LIN {X 0,Y 361.991,Z 217.011,A -85,B 0,C 180,E1 -12946.527,E2 -12946.527} C_VEL
LIN {X 0,Y 362.024,Z 217.007,A -85,B 0,C 180,E1 -12949.938,E2 -12949.938} C_VEL
LIN {X 0,Y 362.155,Z 216.995,A -85,B 0,C 180,E1 -12953.313,E2 -12953.313} C_VEL
LIN {X 0,Y 362.275,Z 216.981,A -85,B 0,C 180,E1 -12957.776,E2 -12957.776} C_VEL
LIN {X 0,Y 362.421,Z 216.956,A -85,B 0,C 180,E1 -12960,E2 -12960} C_VEL
LIN {X 0,Y 362.275,Z 216.984,A -85,B 0,C 180,E1 -12962.223,E2 -12962.223} C_VEL
LIN {X 0,Y 362.155,Z 217,A -85,B 0,C 180,E1 -12966.686,E2 -12966.686} C_VEL
LIN {X 0,Y 362.024,Z 217.013,A -85,B 0,C 180,E1 -12970.062,E2 -12970.062} C_VEL
LIN {X 0,Y 361.99,Z 217.014,A -85,B 0,C 180,E1 -12973.899,E2 -12973.899} C_VEL
LIN {X 0,Y 361.96,Z 217.016,A -85,B 0,C 180,E1 -12977.939,E2 -12977.939} C_VEL
LIN {X 0,Y 361.885,Z 217.026,A -85,B 0,C 180,E1 -12981.653,E2 -12981.653} C_VEL
LIN {X 0,Y 361.921,Z 217.022,A -85,B 0,C 180,E1 -12985.29,E2 -12985.29} C_VEL
LIN {X 0,Y 361.916,Z 217.03,A -85,B 0,C 180,E1 -12987.778,E2 -12987.778} C_VEL
LIN {X 0,Y 361.853,Z 217.036,A -85,B 0,C 180,E1 -12991.628,E2 -12991.628} C_VEL
LIN {X 0,Y 361.868,Z 217.032,A -85,B 0,C 180,E1 -12995.345,E2 -12995.345} C_VEL
LIN {X 0,Y 361.864,Z 217.028,A -85,B 0,C 180,E1 -12999.027,E2 -12999.027} C_VEL
LIN {X 0,Y 361.831,Z 217.039,A -85,B 0,C 180,E1 -13002.829,E2 -13002.829} C_VEL
LIN {X 0,Y 361.821,Z 217.04,A -85,B 0,C 180,E1 -13005.946,E2 -13005.946} C_VEL
LIN {X 0,Y 361.869,Z 217.033,A -85,B 0,C 180,E1 -13009.238,E2 -13009.238} C_VEL
LIN {X 0,Y 361.862,Z 217.11,A -85,B 0,C 180,E1 -13012.901,E2 -13012.901} C_VEL
LIN {X 0,Y 365.155,Z 229.037,A -85,B 0,C 180,E1 -13015.853,E2 -13015.853} C_VEL
LIN {X 0,Y 367.968,Z 240.182,A -85,B 0,C 180,E1 -13018.43,E2 -13018.43} C_VEL
LIN {X 0,Y 374.958,Z 256.162,A -85,B 0,C 180,E1 -13019.427,E2 -13019.427} C_VEL
LIN {X 0,Y 380.018,Z 282.754,A -85,B 0,C 180,E1 -13020.44,E2 -13020.44} C_VEL
LIN {X 0,Y 377.652,Z 382.363,A -85,B 0,C 180,E1 -13022.35,E2 -13022.35} C_VEL
LIN {X 0,Y 376.822,Z 408.501,A -85,B 0,C 180,E1 -13022.886,E2 -13022.886} C_VEL
LIN {X 0,Y 375.878,Z 423.941,A -85,B 0,C 180,E1 -13023.413,E2 -13023.413} C_VEL
LIN {X 0,Y 374.672,Z 437.728,A -85,B 0,C 180,E1 -13024.07,E2 -13024.07} C_VEL
LIN {X 0,Y 373.299,Z 451.151,A -85,B 0,C 180,E1 -13024.913,E2 -13024.913} C_VEL
LIN {X 0,Y 371.548,Z 464.972,A -85,B 0,C 180,E1 -13026.004,E2 -13026.004} C_VEL
LIN {X 0,Y 369.648,Z 478.71,A -85,B 0,C 180,E1 -13027.356,E2 -13027.356} C_VEL
LIN {X 0,Y 367.728,Z 491.149,A -85,B 0,C 180,E1 -13028.855,E2 -13028.855} C_VEL
LIN {X 0,Y 366.079,Z 502.385,A -85,B 0,C 180,E1 -13030.499,E2 -13030.499} C_VEL
LIN {X 0,Y 364.428,Z 512.768,A -85,B 0,C 180,E1 -13032.318,E2 -13032.318} C_VEL
LIN {X 0,Y 363.095,Z 522.038,A -85,B 0,C 180,E1 -13034.278,E2 -13034.278} C_VEL
LIN {X 0,Y 361.936,Z 530.768,A -85,B 0,C 180,E1 -13036.526,E2 -13036.526} C_VEL
LIN {X 0,Y 361.133,Z 537.778,A -85,B 0,C 180,E1 -13038.778,E2 -13038.778} C_VEL
LIN {X 0,Y 360.628,Z 543.293,A -85,B 0,C 180,E1 -13041.031,E2 -13041.031} C_VEL
LIN {X 0,Y 360.386,Z 547.465,A -85,B 0,C 180,E1 -13043.281,E2 -13043.281} C_VEL
LIN {X 0,Y 360.299,Z 550.391,A -85,B 0,C 180,E1 -13045.525,E2 -13045.525} C_VEL
LIN {X 0,Y 360.254,Z 552.136,A -85,B 0,C 180,E1 -13047.764,E2 -13047.764} C_VEL
LIN {X 0,Y 360.357,Z 552.736,A -85,B 0,C 180,E1 -13050,E2 -13050} C_VEL
LIN {X 0,Y 360.255,Z 552.129,A -85,B 0,C 180,E1 -13052.236,E2 -13052.236} C_VEL
LIN {X 0,Y 360.3,Z 550.375,A -85,B 0,C 180,E1 -13054.475,E2 -13054.475} C_VEL
LIN {X 0,Y 360.386,Z 547.445,A -85,B 0,C 180,E1 -13056.719,E2 -13056.719} C_VEL
LIN {X 0,Y 360.628,Z 543.272,A -85,B 0,C 180,E1 -13058.969,E2 -13058.969} C_VEL
LIN {X 0,Y 361.132,Z 537.746,A -85,B 0,C 180,E1 -13061.222,E2 -13061.222} C_VEL
LIN {X 0,Y 361.906,Z 530.719,A -85,B 0,C 180,E1 -13063.475,E2 -13063.475} C_VEL
LIN {X 0,Y 363.096,Z 521.982,A -85,B 0,C 180,E1 -13065.722,E2 -13065.722} C_VEL
LIN {X 0,Y 364.436,Z 512.704,A -85,B 0,C 180,E1 -13067.682,E2 -13067.682} C_VEL
LIN {X 0,Y 365.907,Z 503.649,A -85,B 0,C 180,E1 -13069.284,E2 -13069.284} C_VEL
LIN {X 0,Y 367.612,Z 492.084,A -85,B 0,C 180,E1 -13071.005,E2 -13071.005} C_VEL
LIN {X 0,Y 369.463,Z 479.824,A -85,B 0,C 180,E1 -13072.508,E2 -13072.508} C_VEL
LIN {X 0,Y 371.154,Z 467.779,A -85,B 0,C 180,E1 -13073.726,E2 -13073.726} C_VEL
LIN {X 0,Y 372.912,Z 454.014,A -85,B 0,C 180,E1 -13074.865,E2 -13074.865} C_VEL
LIN {X 0,Y 374.41,Z 440.215,A -85,B 0,C 180,E1 -13075.771,E2 -13075.771} C_VEL
LIN {X 0,Y 375.675,Z 425.49,A -85,B 0,C 180,E1 -13076.513,E2 -13076.513} C_VEL
LIN {X 0,Y 376.707,Z 410.344,A -85,B 0,C 180,E1 -13077.048,E2 -13077.048} C_VEL
LIN {X 0,Y 377.405,Z 390.605,A -85,B 0,C 180,E1 -13077.482,E2 -13077.482} C_VEL
LIN {X 0,Y 380.074,Z 283.543,A -85,B 0,C 180,E1 -13079.523,E2 -13079.523} C_VEL
LIN {X 0,Y 375.075,Z 256.666,A -85,B 0,C 180,E1 -13080.534,E2 -13080.534} C_VEL
LIN {X 0,Y 372.927,Z 251.228,A -85,B 0,C 180,E1 -13080.847,E2 -13080.847} C_VEL
LIN {X 0,Y 367.805,Z 239.811,A -85,B 0,C 180,E1 -13081.61,E2 -13081.61} C_VEL
LIN {X 0,Y 364.596,Z 226.834,A -85,B 0,C 180,E1 -13084.654,E2 -13084.654} C_VEL
LIN {X 0,Y 361.875,Z 217.034,A -85,B 0,C 180,E1 -13087.125,E2 -13087.125} C_VEL
LIN {X 0,Y 361.869,Z 217.034,A -85,B 0,C 180,E1 -13090.762,E2 -13090.762} C_VEL
LIN {X 0,Y 361.817,Z 217.039,A -85,B 0,C 180,E1 -13094.367,E2 -13094.367} C_VEL
LIN {X 0,Y 361.851,Z 217.031,A -85,B 0,C 180,E1 -13097.564,E2 -13097.564} C_VEL
LIN {X 0,Y 361.869,Z 217.029,A -85,B 0,C 180,E1 -13100.972,E2 -13100.972} C_VEL
LIN {X 0,Y 361.869,Z 217.026,A -85,B 0,C 180,E1 -13104.655,E2 -13104.655} C_VEL
LIN {X 0,Y 361.853,Z 217.033,A -85,B 0,C 180,E1 -13108.372,E2 -13108.372} C_VEL
LIN {X 0,Y 361.916,Z 217.025,A -85,B 0,C 180,E1 -13112.222,E2 -13112.222} C_VEL
LIN {X 0,Y 361.92,Z 217.026,A -85,B 0,C 180,E1 -13114.709,E2 -13114.709} C_VEL
LIN {X 0,Y 361.854,Z 217.011,A -85,B 0,C 180,E1 -13118.345,E2 -13118.345} C_VEL
LIN {X 0,Y 361.96,Z 217.022,A -85,B 0,C 180,E1 -13122.061,E2 -13122.061} C_VEL
LIN {X 0,Y 361.99,Z 217.017,A -85,B 0,C 180,E1 -13126.101,E2 -13126.101} C_VEL
LIN {X 0,Y 362.024,Z 217.014,A -85,B 0,C 180,E1 -13129.938,E2 -13129.938} C_VEL
LIN {X 0,Y 362.155,Z 216.999,A -85,B 0,C 180,E1 -13133.314,E2 -13133.314} C_VEL
LIN {X 0,Y 362.275,Z 216.984,A -85,B 0,C 180,E1 -13137.777,E2 -13137.777} C_VEL
LIN {X 0,Y 362.421,Z 216.957,A -85,B 0,C 180,E1 -13140,E2 -13140} C_VEL
LIN {X 0,Y 362.275,Z 216.982,A -85,B 0,C 180,E1 -13142.224,E2 -13142.224} C_VEL
LIN {X 0,Y 362.157,Z 216.997,A -85,B 0,C 180,E1 -13146.687,E2 -13146.687} C_VEL
LIN {X 0,Y 362.024,Z 217.013,A -85,B 0,C 180,E1 -13150.062,E2 -13150.062} C_VEL
LIN {X 0,Y 361.991,Z 217.017,A -85,B 0,C 180,E1 -13153.899,E2 -13153.899} C_VEL
LIN {X 0,Y 361.961,Z 217.02,A -85,B 0,C 180,E1 -13157.939,E2 -13157.939} C_VEL
LIN {X 0,Y 361.855,Z 217.035,A -85,B 0,C 180,E1 -13161.655,E2 -13161.655} C_VEL
LIN {X 0,Y 361.921,Z 217.004,A -85,B 0,C 180,E1 -13165.291,E2 -13165.291} C_VEL
LIN {X 0,Y 361.917,Z 217.022,A -85,B 0,C 180,E1 -13167.778,E2 -13167.778} C_VEL
LIN {X 0,Y 361.841,Z 217.035,A -85,B 0,C 180,E1 -13171.286,E2 -13171.286} C_VEL
LIN {X 0,Y 361.849,Z 217.03,A -85,B 0,C 180,E1 -13174.281,E2 -13174.281} C_VEL
LIN {X 0,Y 361.86,Z 217.032,A -85,B 0,C 180,E1 -13177.224,E2 -13177.224} C_VEL
LIN {X 0,Y 361.832,Z 217.038,A -85,B 0,C 180,E1 -13180.756,E2 -13180.756} C_VEL
LIN {X 0,Y 361.832,Z 217.035,A -85,B 0,C 180,E1 -13184.366,E2 -13184.366} C_VEL
LIN {X 0,Y 361.834,Z 217.038,A -85,B 0,C 180,E1 -13187.569,E2 -13187.569} C_VEL
LIN {X 0,Y 361.867,Z 217.027,A -85,B 0,C 180,E1 -13190.974,E2 -13190.974} C_VEL
LIN {X 0,Y 361.872,Z 217.029,A -85,B 0,C 180,E1 -13194.656,E2 -13194.656} C_VEL
LIN {X 0,Y 361.886,Z 217.145,A -85,B 0,C 180,E1 -13196.515,E2 -13196.515} C_VEL
LIN {X 0,Y 363.49,Z 223.101,A -85,B 0,C 180,E1 -13198.071,E2 -13198.071} C_VEL
LIN {X 0,Y 373.982,Z 244.423,A -85,B 0,C 180,E1 -13199.543,E2 -13199.543} C_VEL
LIN {X 0,Y 380.458,Z 259.445,A -85,B 0,C 180,E1 -13200.441,E2 -13200.441} C_VEL
LIN {X 0,Y 378.098,Z 358.781,A -85,B 0,C 180,E1 -13202.348,E2 -13202.348} C_VEL
LIN {X 0,Y 377.231,Z 388.834,A -85,B 0,C 180,E1 -13202.955,E2 -13202.955} C_VEL
LIN {X 0,Y 376.427,Z 403.824,A -85,B 0,C 180,E1 -13203.46,E2 -13203.46} C_VEL
LIN {X 0,Y 375.345,Z 418.287,A -85,B 0,C 180,E1 -13204.156,E2 -13204.156} C_VEL
LIN {X 0,Y 373.919,Z 433.412,A -85,B 0,C 180,E1 -13205.131,E2 -13205.131} C_VEL
LIN {X 0,Y 372.357,Z 446.659,A -85,B 0,C 180,E1 -13206.207,E2 -13206.207} C_VEL
LIN {X 0,Y 370.485,Z 460.122,A -85,B 0,C 180,E1 -13207.557,E2 -13207.557} C_VEL
LIN {X 0,Y 368.608,Z 472.69,A -85,B 0,C 180,E1 -13209.108,E2 -13209.108} C_VEL
LIN {X 0,Y 366.973,Z 483.449,A -85,B 0,C 180,E1 -13210.71,E2 -13210.71} C_VEL
LIN {X 0,Y 365.256,Z 494.245,A -85,B 0,C 180,E1 -13212.648,E2 -13212.648} C_VEL
LIN {X 0,Y 363.79,Z 503.32,A -85,B 0,C 180,E1 -13214.624,E2 -13214.624} C_VEL
LIN {X 0,Y 362.785,Z 510.621,A -85,B 0,C 180,E1 -13216.558,E2 -13216.558} C_VEL
LIN {X 0,Y 361.722,Z 517.558,A -85,B 0,C 180,E1 -13218.797,E2 -13218.797} C_VEL
LIN {X 0,Y 361.116,Z 523.003,A -85,B 0,C 180,E1 -13221.043,E2 -13221.043} C_VEL
LIN {X 0,Y 360.717,Z 527.515,A -85,B 0,C 180,E1 -13223.544,E2 -13223.544} C_VEL
LIN {X 0,Y 360.486,Z 530,A -85,B 0,C 180,E1 -13225.527,E2 -13225.527} C_VEL
LIN {X 0,Y 360.345,Z 531.738,A -85,B 0,C 180,E1 -13227.765,E2 -13227.765} C_VEL
LIN {X 0,Y 360.36,Z 532.344,A -85,B 0,C 180,E1 -13230,E2 -13230} C_VEL
LIN {X 0,Y 360.345,Z 531.784,A -85,B 0,C 180,E1 -13232.235,E2 -13232.235} C_VEL
LIN {X 0,Y 360.482,Z 530.106,A -85,B 0,C 180,E1 -13234.473,E2 -13234.473} C_VEL
LIN {X 0,Y 360.7,Z 527.276,A -85,B 0,C 180,E1 -13236.713,E2 -13236.713} C_VEL
LIN {X 0,Y 361.094,Z 523.222,A -85,B 0,C 180,E1 -13238.957,E2 -13238.957} C_VEL
LIN {X 0,Y 361.701,Z 517.846,A -85,B 0,C 180,E1 -13241.204,E2 -13241.204} C_VEL
LIN {X 0,Y 362.773,Z 510.986,A -85,B 0,C 180,E1 -13243.443,E2 -13243.443} C_VEL
LIN {X 0,Y 363.787,Z 503.616,A -85,B 0,C 180,E1 -13245.404,E2 -13245.404} C_VEL
LIN {X 0,Y 364.592,Z 498.483,A -85,B 0,C 180,E1 -13246.576,E2 -13246.576} C_VEL
LIN {X 0,Y 364.523,Z 495.062,A -85,B 0,C 180,E1 -13247.322,E2 -13247.322} C_VEL
LIN {X 0,Y 362.726,Z 489.389,A -85,B 0,C 180,E1 -13248.566,E2 -13248.566} C_VEL
LIN {X 0,Y 361.004,Z 483.3,A -85,B 0,C 180,E1 -13249.783,E2 -13249.783} C_VEL
LIN {X 0,Y 361.033,Z 479.222,A -85,B 0,C 180,E1 -13250.468,E2 -13250.468} C_VEL
LIN {X 0,Y 362.793,Z 467.979,A -85,B 0,C 180,E1 -13252.044,E2 -13252.044} C_VEL
LIN {X 0,Y 364.555,Z 456.112,A -85,B 0,C 180,E1 -13253.429,E2 -13253.429} C_VEL
LIN {X 0,Y 366.309,Z 443.263,A -85,B 0,C 180,E1 -13254.663,E2 -13254.663} C_VEL
LIN {X 0,Y 367.946,Z 429.165,A -85,B 0,C 180,E1 -13255.755,E2 -13255.755} C_VEL
LIN {X 0,Y 369.365,Z 413.988,A -85,B 0,C 180,E1 -13256.666,E2 -13256.666} C_VEL
LIN {X 0,Y 370.387,Z 399.264,A -85,B 0,C 180,E1 -13257.319,E2 -13257.319} C_VEL
LIN {X 0,Y 371.137,Z 384.589,A -85,B 0,C 180,E1 -13257.756,E2 -13257.756} C_VEL
LIN {X 0,Y 373.829,Z 283.961,A -85,B 0,C 180,E1 -13259.716,E2 -13259.716} C_VEL
LIN {X 0,Y 374.255,Z 261.257,A -85,B 0,C 180,E1 -13260.172,E2 -13260.172} C_VEL
LIN {X 0,Y 367.754,Z 246.374,A -85,B 0,C 180,E1 -13261.099,E2 -13261.099} C_VEL
LIN {X 0,Y 359.371,Z 229.462,A -85,B 0,C 180,E1 -13262.306,E2 -13262.306} C_VEL
LIN {X 0,Y 356.205,Z 223.066,A -85,B 0,C 180,E1 -13262.799,E2 -13262.799} C_VEL
LIN {X 0,Y 354.823,Z 217.911,A -85,B 0,C 180,E1 -13264.28,E2 -13264.28} C_VEL
LIN {X 0,Y 354.804,Z 217.92,A -85,B 0,C 180,E1 -13267.882,E2 -13267.882} C_VEL
LIN {X 0,Y 354.785,Z 217.918,A -85,B 0,C 180,E1 -13271.171,E2 -13271.171} C_VEL
LIN {X 0,Y 354.786,Z 217.914,A -85,B 0,C 180,E1 -13274.51,E2 -13274.51} C_VEL
LIN {X 0,Y 354.796,Z 217.901,A -85,B 0,C 180,E1 -13277.663,E2 -13277.663} C_VEL
LIN {X 0,Y 354.833,Z 217.91,A -85,B 0,C 180,E1 -13280.668,E2 -13280.668} C_VEL
LIN {X 0,Y 354.817,Z 217.907,A -85,B 0,C 180,E1 -13284.3,E2 -13284.3} C_VEL
LIN {X 0,Y 354.781,Z 217.898,A -85,B 0,C 180,E1 -13287.666,E2 -13287.666} C_VEL
LIN {X 0,Y 354.863,Z 217.9,A -85,B 0,C 180,E1 -13290.621,E2 -13290.621} C_VEL
LIN {X 0,Y 354.893,Z 217.897,A -85,B 0,C 180,E1 -13294.172,E2 -13294.172} C_VEL
LIN {X 0,Y 354.828,Z 217.905,A -85,B 0,C 180,E1 -13297.893,E2 -13297.893} C_VEL
LIN {X 0,Y 354.916,Z 217.893,A -85,B 0,C 180,E1 -13301.891,E2 -13301.891} C_VEL
LIN {X 0,Y 354.935,Z 217.887,A -85,B 0,C 180,E1 -13305.981,E2 -13305.981} C_VEL
LIN {X 0,Y 354.971,Z 217.885,A -85,B 0,C 180,E1 -13309.736,E2 -13309.736} C_VEL
LIN {X 0,Y 355.119,Z 217.872,A -85,B 0,C 180,E1 -13313.18,E2 -13313.18} C_VEL
LIN {X 0,Y 355.238,Z 217.858,A -85,B 0,C 180,E1 -13317.732,E2 -13317.732} C_VEL
LIN {X 0,Y 355.391,Z 217.832,A -85,B 0,C 180,E1 -13320,E2 -13320} C_VEL
LIN {X 0,Y 355.238,Z 217.861,A -85,B 0,C 180,E1 -13322.268,E2 -13322.268} C_VEL
LIN {X 0,Y 355.118,Z 217.875,A -85,B 0,C 180,E1 -13326.819,E2 -13326.819} C_VEL
LIN {X 0,Y 354.97,Z 217.893,A -85,B 0,C 180,E1 -13330.264,E2 -13330.264} C_VEL
LIN {X 0,Y 354.935,Z 217.894,A -85,B 0,C 180,E1 -13334.019,E2 -13334.019} C_VEL
LIN {X 0,Y 354.916,Z 217.895,A -85,B 0,C 180,E1 -13338.109,E2 -13338.109} C_VEL
LIN {X 0,Y 354.827,Z 217.906,A -85,B 0,C 180,E1 -13342.106,E2 -13342.106} C_VEL
LIN {X 0,Y 354.892,Z 217.897,A -85,B 0,C 180,E1 -13345.828,E2 -13345.828} C_VEL
LIN {X 0,Y 354.848,Z 217.909,A -85,B 0,C 180,E1 -13349.679,E2 -13349.679} C_VEL
LIN {X 0,Y 354.825,Z 217.906,A -85,B 0,C 180,E1 -13353.683,E2 -13353.683} C_VEL
LIN {X 0,Y 354.792,Z 217.911,A -85,B 0,C 180,E1 -13356.46,E2 -13356.46} C_VEL
LIN {X 0,Y 354.819,Z 217.899,A -85,B 0,C 180,E1 -13359.424,E2 -13359.424} C_VEL
LIN {X 0,Y 354.783,Z 217.917,A -85,B 0,C 180,E1 -13362.868,E2 -13362.868} C_VEL
LIN {X 0,Y 354.77,Z 217.917,A -85,B 0,C 180,E1 -13366.105,E2 -13366.105} C_VEL
LIN {X 0,Y 354.821,Z 217.911,A -85,B 0,C 180,E1 -13369.185,E2 -13369.185} C_VEL
LIN {X 0,Y 354.84,Z 218.074,A -85,B 0,C 180,E1 -13372.312,E2 -13372.312} C_VEL
LIN {X 0,Y 358.139,Z 229.843,A -85,B 0,C 180,E1 -13375.314,E2 -13375.314} C_VEL
LIN {X 0,Y 360.635,Z 239.833,A -85,B 0,C 180,E1 -13377.708,E2 -13377.708} C_VEL
LIN {X 0,Y 369.134,Z 258.831,A -85,B 0,C 180,E1 -13378.955,E2 -13378.955} C_VEL
LIN {X 0,Y 373.847,Z 283.787,A -85,B 0,C 180,E1 -13379.929,E2 -13379.929} C_VEL
LIN {X 0,Y 371.324,Z 383.972,A -85,B 0,C 180,E1 -13381.876,E2 -13381.876} C_VEL
LIN {X 0,Y 370.526,Z 408.314,A -85,B 0,C 180,E1 -13382.386,E2 -13382.386} C_VEL
LIN {X 0,Y 369.537,Z 423.747,A -85,B 0,C 180,E1 -13382.919,E2 -13382.919} C_VEL
LIN {X 0,Y 368.281,Z 437.523,A -85,B 0,C 180,E1 -13383.585,E2 -13383.585} C_VEL
LIN {X 0,Y 366.796,Z 451.504,A -85,B 0,C 180,E1 -13384.48,E2 -13384.48} C_VEL
LIN {X 0,Y 365.028,Z 464.774,A -85,B 0,C 180,E1 -13385.548,E2 -13385.548} C_VEL
LIN {X 0,Y 363.234,Z 477.216,A -85,B 0,C 180,E1 -13386.783,E2 -13386.783} C_VEL
LIN {X 0,Y 361.28,Z 489.877,A -85,B 0,C 180,E1 -13388.309,E2 -13388.309} C_VEL
LIN {X 0,Y 359.49,Z 500.912,A -85,B 0,C 180,E1 -13389.916,E2 -13389.916} C_VEL
LIN {X 0,Y 357.886,Z 511.075,A -85,B 0,C 180,E1 -13391.688,E2 -13391.688} C_VEL
LIN {X 0,Y 356.374,Z 520.597,A -85,B 0,C 180,E1 -13393.679,E2 -13393.679} C_VEL
LIN {X 0,Y 355.071,Z 529.307,A -85,B 0,C 180,E1 -13395.898,E2 -13395.898} C_VEL
LIN {X 0,Y 354.319,Z 535.951,A -85,B 0,C 180,E1 -13397.979,E2 -13397.979} C_VEL
LIN {X 0,Y 353.646,Z 541.836,A -85,B 0,C 180,E1 -13400.275,E2 -13400.275} C_VEL
LIN {X 0,Y 353.434,Z 545.339,A -85,B 0,C 180,E1 -13401.999,E2 -13401.999} C_VEL
LIN {X 0,Y 353.24,Z 548.878,A -85,B 0,C 180,E1 -13404.291,E2 -13404.291} C_VEL
LIN {X 0,Y 353.191,Z 551.208,A -85,B 0,C 180,E1 -13406.578,E2 -13406.578} C_VEL
LIN {X 0,Y 353.213,Z 552.38,A -85,B 0,C 180,E1 -13408.86,E2 -13408.86} C_VEL
LIN {X 0,Y 353.213,Z 552.377,A -85,B 0,C 180,E1 -13411.14,E2 -13411.14} C_VEL
LIN {X 0,Y 353.192,Z 551.195,A -85,B 0,C 180,E1 -13413.422,E2 -13413.422} C_VEL
LIN {X 0,Y 353.276,Z 548.603,A -85,B 0,C 180,E1 -13415.908,E2 -13415.908} C_VEL
LIN {X 0,Y 353.483,Z 544.241,A -85,B 0,C 180,E1 -13418.576,E2 -13418.576} C_VEL
LIN {X 0,Y 353.921,Z 539.043,A -85,B 0,C 180,E1 -13420.874,E2 -13420.874} C_VEL
LIN {X 0,Y 354.694,Z 532.401,A -85,B 0,C 180,E1 -13423.171,E2 -13423.171} C_VEL
LIN {X 0,Y 355.815,Z 524.128,A -85,B 0,C 180,E1 -13425.465,E2 -13425.465} C_VEL
LIN {X 0,Y 357.16,Z 515.309,A -85,B 0,C 180,E1 -13427.462,E2 -13427.462} C_VEL
LIN {X 0,Y 358.679,Z 506.352,A -85,B 0,C 180,E1 -13429.159,E2 -13429.159} C_VEL
LIN {X 0,Y 360.309,Z 495.798,A -85,B 0,C 180,E1 -13430.853,E2 -13430.853} C_VEL
LIN {X 0,Y 362.167,Z 484.331,A -85,B 0,C 180,E1 -13432.385,E2 -13432.385} C_VEL
LIN {X 0,Y 363.993,Z 471.866,A -85,B 0,C 180,E1 -13433.769,E2 -13433.769} C_VEL
LIN {X 0,Y 365.901,Z 458.218,A -85,B 0,C 180,E1 -13434.996,E2 -13434.996} C_VEL
LIN {X 0,Y 367.635,Z 443.594,A -85,B 0,C 180,E1 -13436.04,E2 -13436.04} C_VEL
LIN {X 0,Y 368.968,Z 429.525,A -85,B 0,C 180,E1 -13436.82,E2 -13436.82} C_VEL
LIN {X 0,Y 370.181,Z 413.557,A -85,B 0,C 180,E1 -13437.45,E2 -13437.45} C_VEL
LIN {X 0,Y 370.938,Z 397.546,A -85,B 0,C 180,E1 -13437.849,E2 -13437.849} C_VEL
LIN {X 0,Y 373.655,Z 292.386,A -85,B 0,C 180,E1 -13439.885,E2 -13439.885} C_VEL
LIN {X 0,Y 373.768,Z 283.974,A -85,B 0,C 180,E1 -13440.057,E2 -13440.057} C_VEL
LIN {X 0,Y 369.092,Z 258.68,A -85,B 0,C 180,E1 -13441.034,E2 -13441.034} C_VEL
LIN {X 0,Y 362.263,Z 243.483,A -85,B 0,C 180,E1 -13442.027,E2 -13442.027} C_VEL
LIN {X 0,Y 360.553,Z 239.569,A -85,B 0,C 180,E1 -13442.324,E2 -13442.324} C_VEL
LIN {X 0,Y 357.378,Z 226.863,A -85,B 0,C 180,E1 -13445.399,E2 -13445.399} C_VEL
LIN {X 0,Y 354.807,Z 217.915,A -85,B 0,C 180,E1 -13447.739,E2 -13447.739} C_VEL
LIN {X 0,Y 354.812,Z 217.911,A -85,B 0,C 180,E1 -13451.176,E2 -13451.176} C_VEL
LIN {X 0,Y 354.763,Z 217.916,A -85,B 0,C 180,E1 -13454.506,E2 -13454.506} C_VEL
LIN {X 0,Y 354.808,Z 217.909,A -85,B 0,C 180,E1 -13457.665,E2 -13457.665} C_VEL
LIN {X 0,Y 354.832,Z 217.906,A -85,B 0,C 180,E1 -13460.668,E2 -13460.668} C_VEL
LIN {X 0,Y 354.817,Z 217.904,A -85,B 0,C 180,E1 -13464.3,E2 -13464.3} C_VEL
LIN {X 0,Y 354.793,Z 217.909,A -85,B 0,C 180,E1 -13467.667,E2 -13467.667} C_VEL
LIN {X 0,Y 354.863,Z 217.901,A -85,B 0,C 180,E1 -13470.621,E2 -13470.621} C_VEL
LIN {X 0,Y 354.892,Z 217.903,A -85,B 0,C 180,E1 -13474.172,E2 -13474.172} C_VEL
LIN {X 0,Y 354.81,Z 217.889,A -85,B 0,C 180,E1 -13477.892,E2 -13477.892} C_VEL
LIN {X 0,Y 354.915,Z 217.901,A -85,B 0,C 180,E1 -13481.891,E2 -13481.891} C_VEL
LIN {X 0,Y 354.935,Z 217.896,A -85,B 0,C 180,E1 -13485.981,E2 -13485.981} C_VEL
LIN {X 0,Y 354.97,Z 217.894,A -85,B 0,C 180,E1 -13489.736,E2 -13489.736} C_VEL
LIN {X 0,Y 355.118,Z 217.874,A -85,B 0,C 180,E1 -13493.181,E2 -13493.181} C_VEL
LIN {X 0,Y 355.238,Z 217.861,A -85,B 0,C 180,E1 -13497.732,E2 -13497.732} C_VEL
LIN {X 0,Y 355.391,Z 217.833,A -85,B 0,C 180,E1 -13500,E2 -13500} C_VEL
LIN {X 0,Y 355.238,Z 217.858,A -85,B 0,C 180,E1 -13502.268,E2 -13502.268} C_VEL
LIN {X 0,Y 355.12,Z 217.875,A -85,B 0,C 180,E1 -13506.82,E2 -13506.82} C_VEL
LIN {X 0,Y 354.971,Z 217.891,A -85,B 0,C 180,E1 -13510.264,E2 -13510.264} C_VEL
LIN {X 0,Y 354.936,Z 217.895,A -85,B 0,C 180,E1 -13514.019,E2 -13514.019} C_VEL
LIN {X 0,Y 354.916,Z 217.898,A -85,B 0,C 180,E1 -13518.109,E2 -13518.109} C_VEL
LIN {X 0,Y 354.81,Z 217.911,A -85,B 0,C 180,E1 -13522.108,E2 -13522.108} C_VEL
LIN {X 0,Y 354.893,Z 217.876,A -85,B 0,C 180,E1 -13525.828,E2 -13525.828} C_VEL
LIN {X 0,Y 354.849,Z 217.907,A -85,B 0,C 180,E1 -13529.679,E2 -13529.679} C_VEL
LIN {X 0,Y 354.801,Z 217.908,A -85,B 0,C 180,E1 -13533.703,E2 -13533.703} C_VEL
LIN {X 0,Y 354.794,Z 217.912,A -85,B 0,C 180,E1 -13536.46,E2 -13536.46} C_VEL
LIN {X 0,Y 354.82,Z 217.906,A -85,B 0,C 180,E1 -13539.424,E2 -13539.424} C_VEL
LIN {X 0,Y 354.785,Z 217.915,A -85,B 0,C 180,E1 -13542.868,E2 -13542.868} C_VEL
LIN {X 0,Y 354.773,Z 217.916,A -85,B 0,C 180,E1 -13546.106,E2 -13546.106} C_VEL
LIN {X 0,Y 354.786,Z 217.919,A -85,B 0,C 180,E1 -13549.18,E2 -13549.18} C_VEL
LIN {X 0,Y 354.809,Z 217.915,A -85,B 0,C 180,E1 -13552.402,E2 -13552.402} C_VEL
LIN {X 0,Y 354.857,Z 218.081,A -85,B 0,C 180,E1 -13555.938,E2 -13555.938} C_VEL
LIN {X 0,Y 356.253,Z 223.233,A -85,B 0,C 180,E1 -13557.339,E2 -13557.339} C_VEL
LIN {X 0,Y 367.238,Z 245.255,A -85,B 0,C 180,E1 -13558.936,E2 -13558.936} C_VEL
LIN {X 0,Y 373.323,Z 258.985,A -85,B 0,C 180,E1 -13559.802,E2 -13559.802} C_VEL
LIN {X 0,Y 374.284,Z 261.371,A -85,B 0,C 180,E1 -13559.94,E2 -13559.94} C_VEL
LIN {X 0,Y 371.58,Z 369.725,A -85,B 0,C 180,E1 -13562.05,E2 -13562.05} C_VEL
LIN {X 0,Y 370.898,Z 390.19,A -85,B 0,C 180,E1 -13562.493,E2 -13562.493} C_VEL
LIN {X 0,Y 370.056,Z 404.688,A -85,B 0,C 180,E1 -13562.999,E2 -13562.999} C_VEL
LIN {X 0,Y 368.925,Z 419.126,A -85,B 0,C 180,E1 -13563.714,E2 -13563.714} C_VEL
LIN {X 0,Y 367.503,Z 433.618,A -85,B 0,C 180,E1 -13564.667,E2 -13564.667} C_VEL
LIN {X 0,Y 365.844,Z 446.866,A -85,B 0,C 180,E1 -13565.757,E2 -13565.757} C_VEL
LIN {X 0,Y 363.925,Z 460.327,A -85,B 0,C 180,E1 -13567.13,E2 -13567.13} C_VEL
LIN {X 0,Y 362.112,Z 471.985,A -85,B 0,C 180,E1 -13568.58,E2 -13568.58} C_VEL
LIN {X 0,Y 360.565,Z 481.886,A -85,B 0,C 180,E1 -13570.056,E2 -13570.056} C_VEL
LIN {X 0,Y 358.93,Z 491.525,A -85,B 0,C 180,E1 -13571.743,E2 -13571.743} C_VEL
LIN {X 0,Y 357.348,Z 500.969,A -85,B 0,C 180,E1 -13573.725,E2 -13573.725} C_VEL
LIN {X 0,Y 356.048,Z 508.829,A -85,B 0,C 180,E1 -13575.716,E2 -13575.716} C_VEL
LIN {X 0,Y 355.273,Z 514.49,A -85,B 0,C 180,E1 -13577.432,E2 -13577.432} C_VEL
LIN {X 0,Y 354.364,Z 520.659,A -85,B 0,C 180,E1 -13579.718,E2 -13579.718} C_VEL
LIN {X 0,Y 353.838,Z 525.419,A -85,B 0,C 180,E1 -13582.008,E2 -13582.008} C_VEL
LIN {X 0,Y 353.511,Z 528.906,A -85,B 0,C 180,E1 -13584.295,E2 -13584.295} C_VEL
LIN {X 0,Y 353.292,Z 531.212,A -85,B 0,C 180,E1 -13586.579,E2 -13586.579} C_VEL
LIN {X 0,Y 353.25,Z 532.388,A -85,B 0,C 180,E1 -13588.86,E2 -13588.86} C_VEL
LIN {X 0,Y 353.25,Z 532.403,A -85,B 0,C 180,E1 -13591.14,E2 -13591.14} C_VEL
LIN {X 0,Y 353.291,Z 531.287,A -85,B 0,C 180,E1 -13593.421,E2 -13593.421} C_VEL
LIN {X 0,Y 353.491,Z 529.04,A -85,B 0,C 180,E1 -13595.705,E2 -13595.705} C_VEL
LIN {X 0,Y 353.807,Z 525.608,A -85,B 0,C 180,E1 -13597.993,E2 -13597.993} C_VEL
LIN {X 0,Y 354.353,Z 520.907,A -85,B 0,C 180,E1 -13600.282,E2 -13600.282} C_VEL
LIN {X 0,Y 355.263,Z 514.812,A -85,B 0,C 180,E1 -13602.568,E2 -13602.568} C_VEL
LIN {X 0,Y 356.166,Z 508.078,A -85,B 0,C 180,E1 -13604.605,E2 -13604.605} C_VEL
LIN {X 0,Y 357.707,Z 498.952,A -85,B 0,C 180,E1 -13606.845,E2 -13606.845} C_VEL
LIN {X 0,Y 359.374,Z 489.086,A -85,B 0,C 180,E1 -13608.824,E2 -13608.824} C_VEL
LIN {X 0,Y 361.033,Z 479.222,A -85,B 0,C 180,E1 -13610.468,E2 -13610.468} C_VEL
LIN {X 0,Y 361.092,Z 475.079,A -85,B 0,C 180,E1 -13611.137,E2 -13611.137} C_VEL
LIN {X 0,Y 359.505,Z 468.236,A -85,B 0,C 180,E1 -13612.25,E2 -13612.25} C_VEL
LIN {X 0,Y 357.951,Z 461.059,A -85,B 0,C 180,E1 -13613.308,E2 -13613.308} C_VEL
LIN {X 0,Y 358.047,Z 456.333,A -85,B 0,C 180,E1 -13613.878,E2 -13613.878} C_VEL
LIN {X 0,Y 359.874,Z 443.458,A -85,B 0,C 180,E1 -13615.135,E2 -13615.135} C_VEL
LIN {X 0,Y 361.556,Z 429.359,A -85,B 0,C 180,E1 -13616.245,E2 -13616.245} C_VEL
LIN {X 0,Y 363.03,Z 414.201,A -85,B 0,C 180,E1 -13617.168,E2 -13617.168} C_VEL
LIN {X 0,Y 364.1,Z 399.452,A -85,B 0,C 180,E1 -13617.831,E2 -13617.831} C_VEL
LIN {X 0,Y 364.894,Z 384.768,A -85,B 0,C 180,E1 -13618.273,E2 -13618.273} C_VEL
LIN {X 0,Y 367.697,Z 283.222,A -85,B 0,C 180,E1 -13620.283,E2 -13620.283} C_VEL
LIN {X 0,Y 368.095,Z 263.183,A -85,B 0,C 180,E1 -13620.692,E2 -13620.692} C_VEL
LIN {X 0,Y 361.25,Z 247.597,A -85,B 0,C 180,E1 -13621.7,E2 -13621.7} C_VEL
LIN {X 0,Y 351.012,Z 227.221,A -85,B 0,C 180,E1 -13623.233,E2 -13623.233} C_VEL
LIN {X 0,Y 348.983,Z 223.307,A -85,B 0,C 180,E1 -13623.565,E2 -13623.565} C_VEL
LIN {X 0,Y 347.778,Z 218.793,A -85,B 0,C 180,E1 -13624.899,E2 -13624.899} C_VEL
LIN {X 0,Y 347.75,Z 218.793,A -85,B 0,C 180,E1 -13628.792,E2 -13628.792} C_VEL
LIN {X 0,Y 347.748,Z 218.794,A -85,B 0,C 180,E1 -13631.829,E2 -13631.829} C_VEL
LIN {X 0,Y 347.763,Z 218.791,A -85,B 0,C 180,E1 -13635.016,E2 -13635.016} C_VEL
LIN {X 0,Y 347.758,Z 218.782,A -85,B 0,C 180,E1 -13638.394,E2 -13638.394} C_VEL
LIN {X 0,Y 347.772,Z 218.772,A -85,B 0,C 180,E1 -13642.01,E2 -13642.01} C_VEL
LIN {X 0,Y 347.74,Z 218.794,A -85,B 0,C 180,E1 -13645.535,E2 -13645.535} C_VEL
LIN {X 0,Y 347.759,Z 218.775,A -85,B 0,C 180,E1 -13649.653,E2 -13649.653} C_VEL
LIN {X 0,Y 347.847,Z 218.78,A -85,B 0,C 180,E1 -13652.744,E2 -13652.744} C_VEL
LIN {X 0,Y 347.782,Z 218.787,A -85,B 0,C 180,E1 -13656.161,E2 -13656.161} C_VEL
LIN {X 0,Y 347.806,Z 218.784,A -85,B 0,C 180,E1 -13659.909,E2 -13659.909} C_VEL
LIN {X 0,Y 347.859,Z 218.773,A -85,B 0,C 180,E1 -13662.359,E2 -13662.359} C_VEL
LIN {X 0,Y 347.891,Z 218.765,A -85,B 0,C 180,E1 -13665.97,E2 -13665.97} C_VEL
LIN {X 0,Y 347.921,Z 218.764,A -85,B 0,C 180,E1 -13669.525,E2 -13669.525} C_VEL
LIN {X 0,Y 348.085,Z 218.75,A -85,B 0,C 180,E1 -13673.042,E2 -13673.042} C_VEL
LIN {X 0,Y 348.2,Z 218.734,A -85,B 0,C 180,E1 -13677.686,E2 -13677.686} C_VEL
LIN {X 0,Y 348.34,Z 218.71,A -85,B 0,C 180,E1 -13680,E2 -13680} C_VEL
LIN {X 0,Y 348.2,Z 218.738,A -85,B 0,C 180,E1 -13682.313,E2 -13682.313} C_VEL
LIN {X 0,Y 348.084,Z 218.75,A -85,B 0,C 180,E1 -13686.958,E2 -13686.958} C_VEL
LIN {X 0,Y 347.921,Z 218.774,A -85,B 0,C 180,E1 -13690.474,E2 -13690.474} C_VEL
LIN {X 0,Y 347.891,Z 218.772,A -85,B 0,C 180,E1 -13694.15,E2 -13694.15} C_VEL
LIN {X 0,Y 347.884,Z 218.772,A -85,B 0,C 180,E1 -13698.291,E2 -13698.291} C_VEL
LIN {X 0,Y 347.781,Z 218.782,A -85,B 0,C 180,E1 -13701.635,E2 -13701.635} C_VEL
LIN {X 0,Y 347.805,Z 218.78,A -85,B 0,C 180,E1 -13705.109,E2 -13705.109} C_VEL
LIN {X 0,Y 347.806,Z 218.787,A -85,B 0,C 180,E1 -13707.694,E2 -13707.694} C_VEL
LIN {X 0,Y 347.764,Z 218.792,A -85,B 0,C 180,E1 -13710.346,E2 -13710.346} C_VEL
LIN {X 0,Y 347.742,Z 218.792,A -85,B 0,C 180,E1 -13714.044,E2 -13714.044} C_VEL
LIN {X 0,Y 347.756,Z 218.79,A -85,B 0,C 180,E1 -13717.321,E2 -13717.321} C_VEL
LIN {X 0,Y 347.726,Z 218.773,A -85,B 0,C 180,E1 -13720.298,E2 -13720.298} C_VEL
LIN {X 0,Y 347.718,Z 218.798,A -85,B 0,C 180,E1 -13723.409,E2 -13723.409} C_VEL
LIN {X 0,Y 347.728,Z 218.794,A -85,B 0,C 180,E1 -13726.686,E2 -13726.686} C_VEL
LIN {X 0,Y 347.754,Z 218.789,A -85,B 0,C 180,E1 -13730.172,E2 -13730.172} C_VEL
LIN {X 0,Y 347.778,Z 218.926,A -85,B 0,C 180,E1 -13731.664,E2 -13731.664} C_VEL
LIN {X 0,Y 351.155,Z 230.761,A -85,B 0,C 180,E1 -13734.78,E2 -13734.78} C_VEL
LIN {X 0,Y 353.376,Z 239.64,A -85,B 0,C 180,E1 -13736.962,E2 -13736.962} C_VEL
LIN {X 0,Y 362.442,Z 259.465,A -85,B 0,C 180,E1 -13738.335,E2 -13738.335} C_VEL
LIN {X 0,Y 363.557,Z 262.526,A -85,B 0,C 180,E1 -13738.512,E2 -13738.512} C_VEL
LIN {X 0,Y 367.695,Z 284.984,A -85,B 0,C 180,E1 -13739.403,E2 -13739.403} C_VEL
LIN {X 0,Y 364.834,Z 392.743,A -85,B 0,C 180,E1 -13741.526,E2 -13741.526} C_VEL
LIN {X 0,Y 364.127,Z 410.408,A -85,B 0,C 180,E1 -13741.937,E2 -13741.937} C_VEL
LIN {X 0,Y 363.028,Z 425.844,A -85,B 0,C 180,E1 -13742.51,E2 -13742.51} C_VEL
LIN {X 0,Y 361.7,Z 439.593,A -85,B 0,C 180,E1 -13743.222,E2 -13743.222} C_VEL
LIN {X 0,Y 360.156,Z 453.215,A -85,B 0,C 180,E1 -13744.14,E2 -13744.14} C_VEL
LIN {X 0,Y 358.34,Z 466.088,A -85,B 0,C 180,E1 -13745.215,E2 -13745.215} C_VEL
LIN {X 0,Y 356.305,Z 479.526,A -85,B 0,C 180,E1 -13746.612,E2 -13746.612} C_VEL
LIN {X 0,Y 354.239,Z 491.767,A -85,B 0,C 180,E1 -13748.162,E2 -13748.162} C_VEL
LIN {X 0,Y 352.398,Z 503.099,A -85,B 0,C 180,E1 -13749.905,E2 -13749.905} C_VEL
LIN {X 0,Y 350.808,Z 512.367,A -85,B 0,C 180,E1 -13751.608,E2 -13751.608} C_VEL
LIN {X 0,Y 349.298,Z 521.636,A -85,B 0,C 180,E1 -13753.64,E2 -13753.64} C_VEL
LIN {X 0,Y 347.955,Z 530.364,A -85,B 0,C 180,E1 -13755.974,E2 -13755.974} C_VEL
LIN {X 0,Y 347.099,Z 537.375,A -85,B 0,C 180,E1 -13758.318,E2 -13758.318} C_VEL
LIN {X 0,Y 346.507,Z 542.89,A -85,B 0,C 180,E1 -13760.662,E2 -13760.662} C_VEL
LIN {X 0,Y 346.225,Z 547.063,A -85,B 0,C 180,E1 -13763.005,E2 -13763.005} C_VEL
LIN {X 0,Y 346.114,Z 549.99,A -85,B 0,C 180,E1 -13765.341,E2 -13765.341} C_VEL
LIN {X 0,Y 346.073,Z 551.735,A -85,B 0,C 180,E1 -13767.672,E2 -13767.672} C_VEL
LIN {X 0,Y 346.162,Z 552.334,A -85,B 0,C 180,E1 -13770,E2 -13770} C_VEL
LIN {X 0,Y 346.073,Z 551.727,A -85,B 0,C 180,E1 -13772.328,E2 -13772.328} C_VEL
LIN {X 0,Y 346.115,Z 549.972,A -85,B 0,C 180,E1 -13774.659,E2 -13774.659} C_VEL
LIN {X 0,Y 346.225,Z 547.04,A -85,B 0,C 180,E1 -13776.995,E2 -13776.995} C_VEL
LIN {X 0,Y 346.507,Z 542.865,A -85,B 0,C 180,E1 -13779.338,E2 -13779.338} C_VEL
LIN {X 0,Y 347.096,Z 537.339,A -85,B 0,C 180,E1 -13781.682,E2 -13781.682} C_VEL
LIN {X 0,Y 347.897,Z 530.308,A -85,B 0,C 180,E1 -13784.029,E2 -13784.029} C_VEL
LIN {X 0,Y 349.104,Z 522.796,A -85,B 0,C 180,E1 -13786.069,E2 -13786.069} C_VEL
LIN {X 0,Y 350.565,Z 513.742,A -85,B 0,C 180,E1 -13788.103,E2 -13788.103} C_VEL
LIN {X 0,Y 352.168,Z 504.51,A -85,B 0,C 180,E1 -13789.831,E2 -13789.831} C_VEL
LIN {X 0,Y 353.954,Z 493.633,A -85,B 0,C 180,E1 -13791.551,E2 -13791.551} C_VEL
LIN {X 0,Y 355.907,Z 481.769,A -85,B 0,C 180,E1 -13793.107,E2 -13793.107} C_VEL
LIN {X 0,Y 357.923,Z 468.798,A -85,B 0,C 180,E1 -13794.506,E2 -13794.506} C_VEL
LIN {X 0,Y 359.804,Z 455.486,A -85,B 0,C 180,E1 -13795.671,E2 -13795.671} C_VEL
LIN {X 0,Y 361.446,Z 441.616,A -85,B 0,C 180,E1 -13796.642,E2 -13796.642} C_VEL
LIN {X 0,Y 362.828,Z 427.054,A -85,B 0,C 180,E1 -13797.428,E2 -13797.428} C_VEL
LIN {X 0,Y 363.969,Z 412.201,A -85,B 0,C 180,E1 -13797.998,E2 -13797.998} C_VEL
LIN {X 0,Y 364.736,Z 395.535,A -85,B 0,C 180,E1 -13798.404,E2 -13798.404} C_VEL
LIN {X 0,Y 367.706,Z 285.975,A -85,B 0,C 180,E1 -13800.556,E2 -13800.556} C_VEL
LIN {X 0,Y 363.405,Z 261.864,A -85,B 0,C 180,E1 -13801.498,E2 -13801.498} C_VEL
LIN {X 0,Y 356.68,Z 246.767,A -85,B 0,C 180,E1 -13802.509,E2 -13802.509} C_VEL
LIN {X 0,Y 353.333,Z 239.454,A -85,B 0,C 180,E1 -13803.04,E2 -13803.04} C_VEL
LIN {X 0,Y 350.439,Z 228.211,A -85,B 0,C 180,E1 -13805.851,E2 -13805.851} C_VEL
LIN {X 0,Y 347.744,Z 218.795,A -85,B 0,C 180,E1 -13808.397,E2 -13808.397} C_VEL
LIN {X 0,Y 347.763,Z 218.791,A -85,B 0,C 180,E1 -13811.827,E2 -13811.827} C_VEL
LIN {X 0,Y 347.705,Z 218.794,A -85,B 0,C 180,E1 -13815.026,E2 -13815.026} C_VEL
LIN {X 0,Y 347.763,Z 218.788,A -85,B 0,C 180,E1 -13818.393,E2 -13818.393} C_VEL
LIN {X 0,Y 347.773,Z 218.783,A -85,B 0,C 180,E1 -13822.01,E2 -13822.01} C_VEL
LIN {X 0,Y 347.739,Z 218.789,A -85,B 0,C 180,E1 -13825.536,E2 -13825.536} C_VEL
LIN {X 0,Y 347.758,Z 218.789,A -85,B 0,C 180,E1 -13828.302,E2 -13828.302} C_VEL
LIN {X 0,Y 347.8,Z 218.781,A -85,B 0,C 180,E1 -13830.99,E2 -13830.99} C_VEL
LIN {X 0,Y 347.825,Z 218.779,A -85,B 0,C 180,E1 -13833.607,E2 -13833.607} C_VEL
LIN {X 0,Y 347.779,Z 218.782,A -85,B 0,C 180,E1 -13836.161,E2 -13836.161} C_VEL
LIN {X 0,Y 347.799,Z 218.773,A -85,B 0,C 180,E1 -13839.909,E2 -13839.909} C_VEL
LIN {X 0,Y 347.859,Z 218.777,A -85,B 0,C 180,E1 -13842.359,E2 -13842.359} C_VEL
LIN {X 0,Y 347.89,Z 218.774,A -85,B 0,C 180,E1 -13845.971,E2 -13845.971} C_VEL
LIN {X 0,Y 347.921,Z 218.774,A -85,B 0,C 180,E1 -13849.526,E2 -13849.526} C_VEL
LIN {X 0,Y 348.084,Z 218.749,A -85,B 0,C 180,E1 -13853.042,E2 -13853.042} C_VEL
LIN {X 0,Y 348.2,Z 218.738,A -85,B 0,C 180,E1 -13857.687,E2 -13857.687} C_VEL
LIN {X 0,Y 348.34,Z 218.711,A -85,B 0,C 180,E1 -13860,E2 -13860} C_VEL
LIN {X 0,Y 348.201,Z 218.735,A -85,B 0,C 180,E1 -13862.314,E2 -13862.314} C_VEL
LIN {X 0,Y 348.086,Z 218.752,A -85,B 0,C 180,E1 -13866.958,E2 -13866.958} C_VEL
LIN {X 0,Y 347.921,Z 218.77,A -85,B 0,C 180,E1 -13870.475,E2 -13870.475} C_VEL
LIN {X 0,Y 347.892,Z 218.773,A -85,B 0,C 180,E1 -13874.15,E2 -13874.15} C_VEL
LIN {X 0,Y 347.884,Z 218.774,A -85,B 0,C 180,E1 -13878.29,E2 -13878.29} C_VEL
LIN {X 0,Y 347.762,Z 218.791,A -85,B 0,C 180,E1 -13881.627,E2 -13881.627} C_VEL
LIN {X 0,Y 347.805,Z 218.764,A -85,B 0,C 180,E1 -13885.109,E2 -13885.109} C_VEL
LIN {X 0,Y 347.807,Z 218.775,A -85,B 0,C 180,E1 -13887.694,E2 -13887.694} C_VEL
LIN {X 0,Y 347.759,Z 218.791,A -85,B 0,C 180,E1 -13890.347,E2 -13890.347} C_VEL
LIN {X 0,Y 347.74,Z 218.788,A -85,B 0,C 180,E1 -13894.465,E2 -13894.465} C_VEL
LIN {X 0,Y 347.77,Z 218.787,A -85,B 0,C 180,E1 -13897.989,E2 -13897.989} C_VEL
LIN {X 0,Y 347.747,Z 218.786,A -85,B 0,C 180,E1 -13901.831,E2 -13901.831} C_VEL
LIN {X 0,Y 347.763,Z 218.791,A -85,B 0,C 180,E1 -13905.017,E2 -13905.017} C_VEL
LIN {X 0,Y 347.748,Z 218.793,A -85,B 0,C 180,E1 -13908.398,E2 -13908.398} C_VEL
LIN {X 0,Y 347.774,Z 218.788,A -85,B 0,C 180,E1 -13912.012,E2 -13912.012} C_VEL
LIN {X 0,Y 347.789,Z 218.824,A -85,B 0,C 180,E1 -13915.278,E2 -13915.278} C_VEL
LIN {X 0,Y 349.087,Z 223.575,A -85,B 0,C 180,E1 -13916.584,E2 -13916.584} C_VEL
LIN {X 0,Y 359.069,Z 243.219,A -85,B 0,C 180,E1 -13918.093,E2 -13918.093} C_VEL
LIN {X 0,Y 365.984,Z 258.223,A -85,B 0,C 180,E1 -13919.108,E2 -13919.108} C_VEL
LIN {X 0,Y 368.151,Z 263.385,A -85,B 0,C 180,E1 -13919.426,E2 -13919.426} C_VEL
LIN {X 0,Y 365.165,Z 375.311,A -85,B 0,C 180,E1 -13921.632,E2 -13921.632} C_VEL
LIN {X 0,Y 364.493,Z 392.686,A -85,B 0,C 180,E1 -13922.045,E2 -13922.045} C_VEL
LIN {X 0,Y 363.577,Z 407.445,A -85,B 0,C 180,E1 -13922.608,E2 -13922.608} C_VEL
LIN {X 0,Y 362.366,Z 421.558,A -85,B 0,C 180,E1 -13923.355,E2 -13923.355} C_VEL
LIN {X 0,Y 360.863,Z 435.586,A -85,B 0,C 180,E1 -13924.322,E2 -13924.322} C_VEL
LIN {X 0,Y 359.161,Z 448.501,A -85,B 0,C 180,E1 -13925.43,E2 -13925.43} C_VEL
LIN {X 0,Y 357.194,Z 461.701,A -85,B 0,C 180,E1 -13926.827,E2 -13926.827} C_VEL
LIN {X 0,Y 355.279,Z 473.39,A -85,B 0,C 180,E1 -13928.331,E2 -13928.331} C_VEL
LIN {X 0,Y 353.547,Z 483.859,A -85,B 0,C 180,E1 -13929.947,E2 -13929.947} C_VEL
LIN {X 0,Y 351.645,Z 494.654,A -85,B 0,C 180,E1 -13931.954,E2 -13931.954} C_VEL
LIN {X 0,Y 350.074,Z 503.612,A -85,B 0,C 180,E1 -13933.976,E2 -13933.976} C_VEL
LIN {X 0,Y 348.898,Z 511.029,A -85,B 0,C 180,E1 -13936.012,E2 -13936.012} C_VEL
LIN {X 0,Y 347.727,Z 517.965,A -85,B 0,C 180,E1 -13938.34,E2 -13938.34} C_VEL
LIN {X 0,Y 347.062,Z 523.408,A -85,B 0,C 180,E1 -13940.677,E2 -13940.677} C_VEL
LIN {X 0,Y 346.614,Z 527.516,A -85,B 0,C 180,E1 -13943.012,E2 -13943.012} C_VEL
LIN {X 0,Y 346.338,Z 530.403,A -85,B 0,C 180,E1 -13945.344,E2 -13945.344} C_VEL
LIN {X 0,Y 346.157,Z 532.14,A -85,B 0,C 180,E1 -13947.673,E2 -13947.673} C_VEL
LIN {X 0,Y 346.166,Z 532.745,A -85,B 0,C 180,E1 -13950,E2 -13950} C_VEL
LIN {X 0,Y 346.157,Z 532.185,A -85,B 0,C 180,E1 -13952.327,E2 -13952.327} C_VEL
LIN {X 0,Y 346.333,Z 530.507,A -85,B 0,C 180,E1 -13954.656,E2 -13954.656} C_VEL
LIN {X 0,Y 346.55,Z 527.677,A -85,B 0,C 180,E1 -13956.989,E2 -13956.989} C_VEL
LIN {X 0,Y 347.05,Z 523.622,A -85,B 0,C 180,E1 -13959.323,E2 -13959.323} C_VEL
LIN {X 0,Y 347.709,Z 518.247,A -85,B 0,C 180,E1 -13961.661,E2 -13961.661} C_VEL
LIN {X 0,Y 348.873,Z 511.388,A -85,B 0,C 180,E1 -13963.989,E2 -13963.989} C_VEL
LIN {X 0,Y 350.032,Z 504.015,A -85,B 0,C 180,E1 -13966.026,E2 -13966.026} C_VEL
LIN {X 0,Y 351.589,Z 495.125,A -85,B 0,C 180,E1 -13968.049,E2 -13968.049} C_VEL
LIN {X 0,Y 353.124,Z 486.059,A -85,B 0,C 180,E1 -13969.775,E2 -13969.775} C_VEL
LIN {X 0,Y 354.896,Z 475.621,A -85,B 0,C 180,E1 -13971.449,E2 -13971.449} C_VEL
LIN {X 0,Y 356.9,Z 463.671,A -85,B 0,C 180,E1 -13973.039,E2 -13973.039} C_VEL
LIN {X 0,Y 358.047,Z 456.333,A -85,B 0,C 180,E1 -13973.878,E2 -13973.878} C_VEL
LIN {X 0,Y 358.163,Z 451.536,A -85,B 0,C 180,E1 -13974.428,E2 -13974.428} C_VEL
LIN {X 0,Y 356.693,Z 443.688,A -85,B 0,C 180,E1 -13975.374,E2 -13975.374} C_VEL
LIN {X 0,Y 355.157,Z 435.574,A -85,B 0,C 180,E1 -13976.255,E2 -13976.255} C_VEL
LIN {X 0,Y 355.125,Z 430.339,A -85,B 0,C 180,E1 -13976.695,E2 -13976.695} C_VEL
LIN {X 0,Y 356.591,Z 416.091,A -85,B 0,C 180,E1 -13977.596,E2 -13977.596} C_VEL
LIN {X 0,Y 357.738,Z 401.467,A -85,B 0,C 180,E1 -13978.29,E2 -13978.29} C_VEL
LIN {X 0,Y 358.616,Z 386.451,A -85,B 0,C 180,E1 -13978.774,E2 -13978.774} C_VEL
LIN {X 0,Y 361.606,Z 283.055,A -85,B 0,C 180,E1 -13980.856,E2 -13980.856} C_VEL
LIN {X 0,Y 361.99,Z 265.193,A -85,B 0,C 180,E1 -13981.225,E2 -13981.225} C_VEL
LIN {X 0,Y 354.349,Z 248.093,A -85,B 0,C 180,E1 -13982.385,E2 -13982.385} C_VEL
LIN {X 0,Y 345.642,Z 230.939,A -85,B 0,C 180,E1 -13983.731,E2 -13983.731} C_VEL
LIN {X 0,Y 341.786,Z 223.541,A -85,B 0,C 180,E1 -13984.369,E2 -13984.369} C_VEL
LIN {X 0,Y 340.727,Z 219.673,A -85,B 0,C 180,E1 -13985.549,E2 -13985.549} C_VEL
LIN {X 0,Y 340.708,Z 219.675,A -85,B 0,C 180,E1 -13988.385,E2 -13988.385} C_VEL
LIN {X 0,Y 340.696,Z 219.671,A -85,B 0,C 180,E1 -13992.045,E2 -13992.045} C_VEL
LIN {X 0,Y 340.681,Z 219.675,A -85,B 0,C 180,E1 -13995.461,E2 -13995.461} C_VEL
LIN {X 0,Y 340.695,Z 219.663,A -85,B 0,C 180,E1 -13998.692,E2 -13998.692} C_VEL
LIN {X 0,Y 340.735,Z 219.651,A -85,B 0,C 180,E1 -14001.773,E2 -14001.773} C_VEL
LIN {X 0,Y 340.718,Z 219.668,A -85,B 0,C 180,E1 -14005.595,E2 -14005.595} C_VEL
LIN {X 0,Y 340.698,Z 219.647,A -85,B 0,C 180,E1 -14008.955,E2 -14008.955} C_VEL
LIN {X 0,Y 340.774,Z 219.662,A -85,B 0,C 180,E1 -14012.473,E2 -14012.473} C_VEL
LIN {X 0,Y 340.75,Z 219.664,A -85,B 0,C 180,E1 -14015.638,E2 -14015.638} C_VEL
LIN {X 0,Y 340.738,Z 219.666,A -85,B 0,C 180,E1 -14019.473,E2 -14019.473} C_VEL
LIN {X 0,Y 340.851,Z 219.645,A -85,B 0,C 180,E1 -14021.984,E2 -14021.984} C_VEL
LIN {X 0,Y 340.863,Z 219.64,A -85,B 0,C 180,E1 -14025.705,E2 -14025.705} C_VEL
LIN {X 0,Y 340.864,Z 219.644,A -85,B 0,C 180,E1 -14029.306,E2 -14029.306} C_VEL
LIN {X 0,Y 341.054,Z 219.627,A -85,B 0,C 180,E1 -14032.898,E2 -14032.898} C_VEL
LIN {X 0,Y 341.162,Z 219.611,A -85,B 0,C 180,E1 -14037.639,E2 -14037.639} C_VEL
LIN {X 0,Y 341.29,Z 219.588,A -85,B 0,C 180,E1 -14040,E2 -14040} C_VEL
LIN {X 0,Y 341.162,Z 219.615,A -85,B 0,C 180,E1 -14042.361,E2 -14042.361} C_VEL
LIN {X 0,Y 341.052,Z 219.624,A -85,B 0,C 180,E1 -14047.102,E2 -14047.102} C_VEL
LIN {X 0,Y 340.863,Z 219.654,A -85,B 0,C 180,E1 -14050.694,E2 -14050.694} C_VEL
LIN {X 0,Y 340.856,Z 219.65,A -85,B 0,C 180,E1 -14054.325,E2 -14054.325} C_VEL
LIN {X 0,Y 340.831,Z 219.653,A -85,B 0,C 180,E1 -14058.467,E2 -14058.467} C_VEL
LIN {X 0,Y 340.747,Z 219.659,A -85,B 0,C 180,E1 -14061.857,E2 -14061.857} C_VEL
LIN {X 0,Y 340.766,Z 219.656,A -85,B 0,C 180,E1 -14065.665,E2 -14065.665} C_VEL
LIN {X 0,Y 340.736,Z 219.668,A -85,B 0,C 180,E1 -14068.32,E2 -14068.32} C_VEL
LIN {X 0,Y 340.71,Z 219.669,A -85,B 0,C 180,E1 -14071.043,E2 -14071.043} C_VEL
LIN {X 0,Y 340.712,Z 219.668,A -85,B 0,C 180,E1 -14075.279,E2 -14075.279} C_VEL
LIN {X 0,Y 340.704,Z 219.667,A -85,B 0,C 180,E1 -14078.386,E2 -14078.386} C_VEL
LIN {X 0,Y 340.694,Z 219.661,A -85,B 0,C 180,E1 -14082.046,E2 -14082.046} C_VEL
LIN {X 0,Y 340.652,Z 219.675,A -85,B 0,C 180,E1 -14086.227,E2 -14086.227} C_VEL
LIN {X 0,Y 340.701,Z 219.668,A -85,B 0,C 180,E1 -14088.694,E2 -14088.694} C_VEL
LIN {X 0,Y 340.732,Z 219.736,A -85,B 0,C 180,E1 -14090.973,E2 -14090.973} C_VEL
LIN {X 0,Y 344.248,Z 232.011,A -85,B 0,C 180,E1 -14094.307,E2 -14094.307} C_VEL
LIN {X 0,Y 346.152,Z 239.564,A -85,B 0,C 180,E1 -14096.184,E2 -14096.184} C_VEL
LIN {X 0,Y 355.307,Z 259.034,A -85,B 0,C 180,E1 -14097.617,E2 -14097.617} C_VEL
LIN {X 0,Y 357.735,Z 265.14,A -85,B 0,C 180,E1 -14098.003,E2 -14098.003} C_VEL
LIN {X 0,Y 361.576,Z 286.182,A -85,B 0,C 180,E1 -14098.859,E2 -14098.859} C_VEL
LIN {X 0,Y 358.519,Z 396.144,A -85,B 0,C 180,E1 -14101.057,E2 -14101.057} C_VEL
LIN {X 0,Y 357.775,Z 412.502,A -85,B 0,C 180,E1 -14101.473,E2 -14101.473} C_VEL
LIN {X 0,Y 356.527,Z 427.94,A -85,B 0,C 180,E1 -14102.085,E2 -14102.085} C_VEL
LIN {X 0,Y 354.984,Z 442.794,A -85,B 0,C 180,E1 -14102.913,E2 -14102.913} C_VEL
LIN {X 0,Y 353.206,Z 456.879,A -85,B 0,C 180,E1 -14103.939,E2 -14103.939} C_VEL
LIN {X 0,Y 351.201,Z 470.178,A -85,B 0,C 180,E1 -14105.151,E2 -14105.151} C_VEL
LIN {X 0,Y 349.158,Z 482.86,A -85,B 0,C 180,E1 -14106.576,E2 -14106.576} C_VEL
LIN {X 0,Y 347.255,Z 493.528,A -85,B 0,C 180,E1 -14108.012,E2 -14108.012} C_VEL
LIN {X 0,Y 345.419,Z 504.391,A -85,B 0,C 180,E1 -14109.765,E2 -14109.765} C_VEL
LIN {X 0,Y 343.76,Z 513.608,A -85,B 0,C 180,E1 -14111.526,E2 -14111.526} C_VEL
LIN {X 0,Y 342.206,Z 522.654,A -85,B 0,C 180,E1 -14113.598,E2 -14113.598} C_VEL
LIN {X 0,Y 340.997,Z 530.163,A -85,B 0,C 180,E1 -14115.681,E2 -14115.681} C_VEL
LIN {X 0,Y 340.082,Z 537.174,A -85,B 0,C 180,E1 -14118.074,E2 -14118.074} C_VEL
LIN {X 0,Y 339.431,Z 542.688,A -85,B 0,C 180,E1 -14120.466,E2 -14120.466} C_VEL
LIN {X 0,Y 339.144,Z 546.862,A -85,B 0,C 180,E1 -14122.858,E2 -14122.858} C_VEL
LIN {X 0,Y 339.019,Z 549.789,A -85,B 0,C 180,E1 -14125.244,E2 -14125.244} C_VEL
LIN {X 0,Y 338.987,Z 551.534,A -85,B 0,C 180,E1 -14127.624,E2 -14127.624} C_VEL
LIN {X 0,Y 339.065,Z 552.134,A -85,B 0,C 180,E1 -14130,E2 -14130} C_VEL
LIN {X 0,Y 338.987,Z 551.526,A -85,B 0,C 180,E1 -14132.376,E2 -14132.376} C_VEL
LIN {X 0,Y 339.019,Z 549.77,A -85,B 0,C 180,E1 -14134.756,E2 -14134.756} C_VEL
LIN {X 0,Y 339.144,Z 546.838,A -85,B 0,C 180,E1 -14137.142,E2 -14137.142} C_VEL
LIN {X 0,Y 339.431,Z 542.661,A -85,B 0,C 180,E1 -14139.534,E2 -14139.534} C_VEL
LIN {X 0,Y 340.078,Z 537.135,A -85,B 0,C 180,E1 -14141.926,E2 -14141.926} C_VEL
LIN {X 0,Y 340.911,Z 530.103,A -85,B 0,C 180,E1 -14144.322,E2 -14144.322} C_VEL
LIN {X 0,Y 342.207,Z 522.592,A -85,B 0,C 180,E1 -14146.402,E2 -14146.402} C_VEL
LIN {X 0,Y 343.77,Z 513.538,A -85,B 0,C 180,E1 -14148.474,E2 -14148.474} C_VEL
LIN {X 0,Y 345.6,Z 503.166,A -85,B 0,C 180,E1 -14150.44,E2 -14150.44} C_VEL
LIN {X 0,Y 347.624,Z 491.467,A -85,B 0,C 180,E1 -14152.276,E2 -14152.276} C_VEL
LIN {X 0,Y 349.769,Z 479.208,A -85,B 0,C 180,E1 -14153.852,E2 -14153.852} C_VEL
LIN {X 0,Y 351.872,Z 465.729,A -85,B 0,C 180,E1 -14155.272,E2 -14155.272} C_VEL
LIN {X 0,Y 353.89,Z 451.454,A -85,B 0,C 180,E1 -14156.474,E2 -14156.474} C_VEL
LIN {X 0,Y 355.607,Z 436.885,A -85,B 0,C 180,E1 -14157.434,E2 -14157.434} C_VEL
LIN {X 0,Y 356.936,Z 423.03,A -85,B 0,C 180,E1 -14158.12,E2 -14158.12} C_VEL
LIN {X 0,Y 357.95,Z 408.56,A -85,B 0,C 180,E1 -14158.632,E2 -14158.632} C_VEL
LIN {X 0,Y 358.784,Z 384.568,A -85,B 0,C 180,E1 -14159.16,E2 -14159.16} C_VEL
LIN {X 0,Y 361.558,Z 286.946,A -85,B 0,C 180,E1 -14161.106,E2 -14161.106} C_VEL
LIN {X 0,Y 357.563,Z 264.304,A -85,B 0,C 180,E1 -14162.012,E2 -14162.012} C_VEL
LIN {X 0,Y 349.748,Z 247.065,A -85,B 0,C 180,E1 -14163.222,E2 -14163.222} C_VEL
LIN {X 0,Y 346.029,Z 239.159,A -85,B 0,C 180,E1 -14163.842,E2 -14163.842} C_VEL
LIN {X 0,Y 343.098,Z 227.967,A -85,B 0,C 180,E1 -14166.742,E2 -14166.742} C_VEL
LIN {X 0,Y 340.716,Z 219.67,A -85,B 0,C 180,E1 -14169.06,E2 -14169.06} C_VEL
LIN {X 0,Y 340.698,Z 219.668,A -85,B 0,C 180,E1 -14172.9,E2 -14172.9} C_VEL
LIN {X 0,Y 340.679,Z 219.668,A -85,B 0,C 180,E1 -14177.096,E2 -14177.096} C_VEL
LIN {X 0,Y 340.705,Z 219.668,A -85,B 0,C 180,E1 -14180.248,E2 -14180.248} C_VEL
LIN {X 0,Y 340.707,Z 219.666,A -85,B 0,C 180,E1 -14183.558,E2 -14183.558} C_VEL
LIN {X 0,Y 340.689,Z 219.667,A -85,B 0,C 180,E1 -14186.153,E2 -14186.153} C_VEL
LIN {X 0,Y 340.769,Z 219.656,A -85,B 0,C 180,E1 -14190.332,E2 -14190.332} C_VEL
LIN {X 0,Y 340.799,Z 219.653,A -85,B 0,C 180,E1 -14193.02,E2 -14193.02} C_VEL
LIN {X 0,Y 340.748,Z 219.663,A -85,B 0,C 180,E1 -14195.638,E2 -14195.638} C_VEL
LIN {X 0,Y 340.727,Z 219.648,A -85,B 0,C 180,E1 -14199.473,E2 -14199.473} C_VEL
LIN {X 0,Y 340.851,Z 219.652,A -85,B 0,C 180,E1 -14201.984,E2 -14201.984} C_VEL
LIN {X 0,Y 340.862,Z 219.652,A -85,B 0,C 180,E1 -14205.705,E2 -14205.705} C_VEL
LIN {X 0,Y 340.863,Z 219.651,A -85,B 0,C 180,E1 -14209.306,E2 -14209.306} C_VEL
LIN {X 0,Y 341.052,Z 219.624,A -85,B 0,C 180,E1 -14212.898,E2 -14212.898} C_VEL
LIN {X 0,Y 341.162,Z 219.615,A -85,B 0,C 180,E1 -14217.639,E2 -14217.639} C_VEL
LIN {X 0,Y 341.29,Z 219.589,A -85,B 0,C 180,E1 -14220,E2 -14220} C_VEL
LIN {X 0,Y 341.162,Z 219.612,A -85,B 0,C 180,E1 -14222.361,E2 -14222.361} C_VEL
LIN {X 0,Y 341.053,Z 219.628,A -85,B 0,C 180,E1 -14227.102,E2 -14227.102} C_VEL
LIN {X 0,Y 340.864,Z 219.65,A -85,B 0,C 180,E1 -14230.694,E2 -14230.694} C_VEL
LIN {X 0,Y 340.856,Z 219.649,A -85,B 0,C 180,E1 -14234.325,E2 -14234.325} C_VEL
LIN {X 0,Y 340.83,Z 219.653,A -85,B 0,C 180,E1 -14238.467,E2 -14238.467} C_VEL
LIN {X 0,Y 340.712,Z 219.668,A -85,B 0,C 180,E1 -14241.842,E2 -14241.842} C_VEL
LIN {X 0,Y 340.766,Z 219.635,A -85,B 0,C 180,E1 -14245.665,E2 -14245.665} C_VEL
LIN {X 0,Y 340.737,Z 219.661,A -85,B 0,C 180,E1 -14248.32,E2 -14248.32} C_VEL
LIN {X 0,Y 340.699,Z 219.668,A -85,B 0,C 180,E1 -14251.045,E2 -14251.045} C_VEL
LIN {X 0,Y 340.713,Z 219.669,A -85,B 0,C 180,E1 -14255.28,E2 -14255.28} C_VEL
LIN {X 0,Y 340.706,Z 219.668,A -85,B 0,C 180,E1 -14258.387,E2 -14258.387} C_VEL
LIN {X 0,Y 340.695,Z 219.664,A -85,B 0,C 180,E1 -14262.046,E2 -14262.046} C_VEL
LIN {X 0,Y 340.681,Z 219.672,A -85,B 0,C 180,E1 -14265.462,E2 -14265.462} C_VEL
LIN {X 0,Y 340.684,Z 219.673,A -85,B 0,C 180,E1 -14268.691,E2 -14268.691} C_VEL
LIN {X 0,Y 340.733,Z 219.662,A -85,B 0,C 180,E1 -14271.774,E2 -14271.774} C_VEL
LIN {X 0,Y 340.747,Z 219.751,A -85,B 0,C 180,E1 -14274.635,E2 -14274.635} C_VEL
LIN {X 0,Y 341.878,Z 223.708,A -85,B 0,C 180,E1 -14275.78,E2 -14275.78} C_VEL
LIN {X 0,Y 352.976,Z 245.268,A -85,B 0,C 180,E1 -14277.518,E2 -14277.518} C_VEL
LIN {X 0,Y 360.586,Z 261.948,A -85,B 0,C 180,E1 -14278.674,E2 -14278.674} C_VEL
LIN {X 0,Y 362.01,Z 265.31,A -85,B 0,C 180,E1 -14278.889,E2 -14278.889} C_VEL
LIN {X 0,Y 358.894,Z 377.323,A -85,B 0,C 180,E1 -14281.13,E2 -14281.13} C_VEL
LIN {X 0,Y 358.255,Z 392.902,A -85,B 0,C 180,E1 -14281.515,E2 -14281.515} C_VEL
LIN {X 0,Y 357.269,Z 407.893,A -85,B 0,C 180,E1 -14282.095,E2 -14282.095} C_VEL
LIN {X 0,Y 356.01,Z 422.142,A -85,B 0,C 180,E1 -14282.867,E2 -14282.867} C_VEL
LIN {X 0,Y 354.49,Z 435.793,A -85,B 0,C 180,E1 -14283.825,E2 -14283.825} C_VEL
LIN {X 0,Y 352.711,Z 448.707,A -85,B 0,C 180,E1 -14284.95,E2 -14284.95} C_VEL
LIN {X 0,Y 350.652,Z 461.907,A -85,B 0,C 180,E1 -14286.369,E2 -14286.369} C_VEL
LIN {X 0,Y 348.619,Z 473.897,A -85,B 0,C 180,E1 -14287.943,E2 -14287.943} C_VEL
LIN {X 0,Y 346.88,Z 484.063,A -85,B 0,C 180,E1 -14289.544,E2 -14289.544} C_VEL
LIN {X 0,Y 344.87,Z 494.859,A -85,B 0,C 180,E1 -14291.587,E2 -14291.587} C_VEL
LIN {X 0,Y 343.207,Z 503.816,A -85,B 0,C 180,E1 -14293.647,E2 -14293.647} C_VEL
LIN {X 0,Y 341.947,Z 511.234,A -85,B 0,C 180,E1 -14295.722,E2 -14295.722} C_VEL
LIN {X 0,Y 341.04,Z 516.568,A -85,B 0,C 180,E1 -14297.504,E2 -14297.504} C_VEL
LIN {X 0,Y 340.148,Z 522.384,A -85,B 0,C 180,E1 -14299.885,E2 -14299.885} C_VEL
LIN {X 0,Y 339.746,Z 525.824,A -85,B 0,C 180,E1 -14301.674,E2 -14301.674} C_VEL
LIN {X 0,Y 339.367,Z 529.309,A -85,B 0,C 180,E1 -14304.057,E2 -14304.057} C_VEL
LIN {X 0,Y 339.145,Z 531.614,A -85,B 0,C 180,E1 -14306.436,E2 -14306.436} C_VEL
LIN {X 0,Y 339.055,Z 532.79,A -85,B 0,C 180,E1 -14308.812,E2 -14308.812} C_VEL
LIN {X 0,Y 339.055,Z 532.804,A -85,B 0,C 180,E1 -14311.188,E2 -14311.188} C_VEL
LIN {X 0,Y 339.143,Z 531.687,A -85,B 0,C 180,E1 -14313.564,E2 -14313.564} C_VEL
LIN {X 0,Y 339.346,Z 529.441,A -85,B 0,C 180,E1 -14315.944,E2 -14315.944} C_VEL
LIN {X 0,Y 339.723,Z 526.008,A -85,B 0,C 180,E1 -14318.326,E2 -14318.326} C_VEL
LIN {X 0,Y 340.322,Z 521.309,A -85,B 0,C 180,E1 -14320.711,E2 -14320.711} C_VEL
LIN {X 0,Y 341.382,Z 515.212,A -85,B 0,C 180,E1 -14323.088,E2 -14323.088} C_VEL
LIN {X 0,Y 342.562,Z 507.54,A -85,B 0,C 180,E1 -14325.468,E2 -14325.468} C_VEL
LIN {X 0,Y 344.087,Z 499.351,A -85,B 0,C 180,E1 -14327.533,E2 -14327.533} C_VEL
LIN {X 0,Y 345.881,Z 489.484,A -85,B 0,C 180,E1 -14329.588,E2 -14329.588} C_VEL
LIN {X 0,Y 347.911,Z 478.178,A -85,B 0,C 180,E1 -14331.523,E2 -14331.523} C_VEL
LIN {X 0,Y 349.976,Z 466.205,A -85,B 0,C 180,E1 -14333.209,E2 -14333.209} C_VEL
LIN {X 0,Y 351.946,Z 453.926,A -85,B 0,C 180,E1 -14334.635,E2 -14334.635} C_VEL
LIN {X 0,Y 353.912,Z 440.497,A -85,B 0,C 180,E1 -14335.904,E2 -14335.904} C_VEL
LIN {X 0,Y 355.125,Z 430.339,A -85,B 0,C 180,E1 -14336.695,E2 -14336.695} C_VEL
LIN {X 0,Y 355.119,Z 425.017,A -85,B 0,C 180,E1 -14337.113,E2 -14337.113} C_VEL
LIN {X 0,Y 353.407,Z 416.399,A -85,B 0,C 180,E1 -14337.863,E2 -14337.863} C_VEL
LIN {X 0,Y 351.668,Z 407.59,A -85,B 0,C 180,E1 -14338.536,E2 -14338.536} C_VEL
LIN {X 0,Y 351.497,Z 401.978,A -85,B 0,C 180,E1 -14338.825,E2 -14338.825} C_VEL
LIN {X 0,Y 352.423,Z 386.63,A -85,B 0,C 180,E1 -14339.328,E2 -14339.328} C_VEL
LIN {X 0,Y 355.528,Z 283.175,A -85,B 0,C 180,E1 -14341.444,E2 -14341.444} C_VEL
LIN {X 0,Y 355.871,Z 267.017,A -85,B 0,C 180,E1 -14341.786,E2 -14341.786} C_VEL
LIN {X 0,Y 348.507,Z 250.805,A -85,B 0,C 180,E1 -14342.935,E2 -14342.935} C_VEL
LIN {X 0,Y 340.486,Z 234.914,A -85,B 0,C 180,E1 -14344.216,E2 -14344.216} C_VEL
LIN {X 0,Y 334.567,Z 223.767,A -85,B 0,C 180,E1 -14345.222,E2 -14345.222} C_VEL
LIN {X 0,Y 333.676,Z 220.544,A -85,B 0,C 180,E1 -14346.224,E2 -14346.224} C_VEL
LIN {X 0,Y 333.644,Z 220.545,A -85,B 0,C 180,E1 -14349.192,E2 -14349.192} C_VEL
LIN {X 0,Y 333.63,Z 220.55,A -85,B 0,C 180,E1 -14352.499,E2 -14352.499} C_VEL
LIN {X 0,Y 333.62,Z 220.551,A -85,B 0,C 180,E1 -14355.959,E2 -14355.959} C_VEL
LIN {X 0,Y 333.651,Z 220.547,A -85,B 0,C 180,E1 -14359.313,E2 -14359.313} C_VEL
LIN {X 0,Y 333.651,Z 220.528,A -85,B 0,C 180,E1 -14362.349,E2 -14362.349} C_VEL
LIN {X 0,Y 333.669,Z 220.549,A -85,B 0,C 180,E1 -14365.341,E2 -14365.341} C_VEL
LIN {X 0,Y 333.698,Z 220.525,A -85,B 0,C 180,E1 -14369.71,E2 -14369.71} C_VEL
LIN {X 0,Y 333.739,Z 220.538,A -85,B 0,C 180,E1 -14372.401,E2 -14372.401} C_VEL
LIN {X 0,Y 333.721,Z 220.541,A -85,B 0,C 180,E1 -14375.09,E2 -14375.09} C_VEL
LIN {X 0,Y 333.674,Z 220.547,A -85,B 0,C 180,E1 -14379.019,E2 -14379.019} C_VEL
LIN {X 0,Y 333.787,Z 220.524,A -85,B 0,C 180,E1 -14381.589,E2 -14381.589} C_VEL
LIN {X 0,Y 333.802,Z 220.52,A -85,B 0,C 180,E1 -14385.576,E2 -14385.576} C_VEL
LIN {X 0,Y 333.827,Z 220.522,A -85,B 0,C 180,E1 -14389.078,E2 -14389.078} C_VEL
LIN {X 0,Y 334.006,Z 220.507,A -85,B 0,C 180,E1 -14392.747,E2 -14392.747} C_VEL
LIN {X 0,Y 333.803,Z 220.522,A -85,B 0,C 180,E1 -14395.169,E2 -14395.169} C_VEL
LIN {X 0,Y 334.099,Z 220.491,A -85,B 0,C 180,E1 -14397.589,E2 -14397.589} C_VEL
LIN {X 0,Y 334.241,Z 220.466,A -85,B 0,C 180,E1 -14400,E2 -14400} C_VEL
LIN {X 0,Y 334.099,Z 220.494,A -85,B 0,C 180,E1 -14402.411,E2 -14402.411} C_VEL
LIN {X 0,Y 334.008,Z 220.504,A -85,B 0,C 180,E1 -14406.039,E2 -14406.039} C_VEL
LIN {X 0,Y 333.951,Z 220.504,A -85,B 0,C 180,E1 -14408.471,E2 -14408.471} C_VEL
LIN {X 0,Y 333.784,Z 220.53,A -85,B 0,C 180,E1 -14412.155,E2 -14412.155} C_VEL
LIN {X 0,Y 333.771,Z 220.536,A -85,B 0,C 180,E1 -14415.886,E2 -14415.886} C_VEL
LIN {X 0,Y 333.79,Z 220.533,A -85,B 0,C 180,E1 -14418.655,E2 -14418.655} C_VEL
LIN {X 0,Y 333.686,Z 220.541,A -85,B 0,C 180,E1 -14422.278,E2 -14422.278} C_VEL
LIN {X 0,Y 333.729,Z 220.535,A -85,B 0,C 180,E1 -14426.247,E2 -14426.247} C_VEL
LIN {X 0,Y 333.706,Z 220.543,A -85,B 0,C 180,E1 -14428.972,E2 -14428.972} C_VEL
LIN {X 0,Y 333.645,Z 220.543,A -85,B 0,C 180,E1 -14432.59,E2 -14432.59} C_VEL
LIN {X 0,Y 333.67,Z 220.541,A -85,B 0,C 180,E1 -14436.14,E2 -14436.14} C_VEL
LIN {X 0,Y 333.641,Z 220.538,A -85,B 0,C 180,E1 -14439.193,E2 -14439.193} C_VEL
LIN {X 0,Y 333.627,Z 220.548,A -85,B 0,C 180,E1 -14442.5,E2 -14442.5} C_VEL
LIN {X 0,Y 333.596,Z 220.555,A -85,B 0,C 180,E1 -14445.956,E2 -14445.956} C_VEL
LIN {X 0,Y 333.653,Z 220.549,A -85,B 0,C 180,E1 -14449.314,E2 -14449.314} C_VEL
LIN {X 0,Y 333.692,Z 220.634,A -85,B 0,C 180,E1 -14450.269,E2 -14450.269} C_VEL
LIN {X 0,Y 337.325,Z 233.373,A -85,B 0,C 180,E1 -14453.836,E2 -14453.836} C_VEL
LIN {X 0,Y 338.836,Z 239.111,A -85,B 0,C 180,E1 -14455.345,E2 -14455.345} C_VEL
LIN {X 0,Y 348.488,Z 259.556,A -85,B 0,C 180,E1 -14456.921,E2 -14456.921} C_VEL
LIN {X 0,Y 351.937,Z 267.659,A -85,B 0,C 180,E1 -14457.476,E2 -14457.476} C_VEL
LIN {X 0,Y 355.493,Z 287.347,A -85,B 0,C 180,E1 -14458.296,E2 -14458.296} C_VEL
LIN {X 0,Y 352.017,Z 403.857,A -85,B 0,C 180,E1 -14460.676,E2 -14460.676} C_VEL
LIN {X 0,Y 351.081,Z 418.975,A -85,B 0,C 180,E1 -14461.164,E2 -14461.164} C_VEL
LIN {X 0,Y 349.537,Z 434.422,A -85,B 0,C 180,E1 -14461.885,E2 -14461.885} C_VEL
LIN {X 0,Y 347.983,Z 448.019,A -85,B 0,C 180,E1 -14462.754,E2 -14462.754} C_VEL
LIN {X 0,Y 346.166,Z 461.013,A -85,B 0,C 180,E1 -14463.796,E2 -14463.796} C_VEL
LIN {X 0,Y 344.071,Z 474.031,A -85,B 0,C 180,E1 -14465.085,E2 -14465.085} C_VEL
LIN {X 0,Y 342.053,Z 486.059,A -85,B 0,C 180,E1 -14466.542,E2 -14466.542} C_VEL
LIN {X 0,Y 339.969,Z 497.201,A -85,B 0,C 180,E1 -14468.155,E2 -14468.155} C_VEL
LIN {X 0,Y 338.148,Z 507.463,A -85,B 0,C 180,E1 -14469.945,E2 -14469.945} C_VEL
LIN {X 0,Y 336.206,Z 517.492,A -85,B 0,C 180,E1 -14472.042,E2 -14472.042} C_VEL
LIN {X 0,Y 334.72,Z 525.828,A -85,B 0,C 180,E1 -14474.16,E2 -14474.16} C_VEL
LIN {X 0,Y 333.512,Z 533.666,A -85,B 0,C 180,E1 -14476.597,E2 -14476.597} C_VEL
LIN {X 0,Y 332.625,Z 539.903,A -85,B 0,C 180,E1 -14479.038,E2 -14479.038} C_VEL
LIN {X 0,Y 332.222,Z 544.735,A -85,B 0,C 180,E1 -14481.484,E2 -14481.484} C_VEL
LIN {X 0,Y 332.007,Z 548.625,A -85,B 0,C 180,E1 -14484.213,E2 -14484.213} C_VEL
LIN {X 0,Y 331.941,Z 550.606,A -85,B 0,C 180,E1 -14486.358,E2 -14486.358} C_VEL
LIN {X 0,Y 331.92,Z 551.777,A -85,B 0,C 180,E1 -14488.787,E2 -14488.787} C_VEL
LIN {X 0,Y 331.92,Z 551.775,A -85,B 0,C 180,E1 -14491.213,E2 -14491.213} C_VEL
LIN {X 0,Y 331.941,Z 550.592,A -85,B 0,C 180,E1 -14493.642,E2 -14493.642} C_VEL
LIN {X 0,Y 331.993,Z 548.253,A -85,B 0,C 180,E1 -14496.076,E2 -14496.076} C_VEL
LIN {X 0,Y 332.222,Z 544.709,A -85,B 0,C 180,E1 -14498.516,E2 -14498.516} C_VEL
LIN {X 0,Y 332.625,Z 539.87,A -85,B 0,C 180,E1 -14500.962,E2 -14500.962} C_VEL
LIN {X 0,Y 333.489,Z 533.614,A -85,B 0,C 180,E1 -14503.404,E2 -14503.404} C_VEL
LIN {X 0,Y 334.557,Z 526.853,A -85,B 0,C 180,E1 -14505.535,E2 -14505.535} C_VEL
LIN {X 0,Y 335.971,Z 518.684,A -85,B 0,C 180,E1 -14507.657,E2 -14507.657} C_VEL
LIN {X 0,Y 337.853,Z 508.898,A -85,B 0,C 180,E1 -14509.757,E2 -14509.757} C_VEL
LIN {X 0,Y 339.701,Z 498.464,A -85,B 0,C 180,E1 -14511.62,E2 -14511.62} C_VEL
LIN {X 0,Y 341.811,Z 487.016,A -85,B 0,C 180,E1 -14513.315,E2 -14513.315} C_VEL
LIN {X 0,Y 343.82,Z 475.183,A -85,B 0,C 180,E1 -14514.773,E2 -14514.773} C_VEL
LIN {X 0,Y 345.917,Z 462.407,A -85,B 0,C 180,E1 -14516.062,E2 -14516.062} C_VEL
LIN {X 0,Y 347.788,Z 449.27,A -85,B 0,C 180,E1 -14517.14,E2 -14517.14} C_VEL
LIN {X 0,Y 349.42,Z 435.425,A -85,B 0,C 180,E1 -14518.043,E2 -14518.043} C_VEL
LIN {X 0,Y 350.833,Z 421.272,A -85,B 0,C 180,E1 -14518.735,E2 -14518.735} C_VEL
LIN {X 0,Y 351.909,Z 406.052,A -85,B 0,C 180,E1 -14519.252,E2 -14519.252} C_VEL
LIN {X 0,Y 355.227,Z 296.106,A -85,B 0,C 180,E1 -14521.506,E2 -14521.506} C_VEL
LIN {X 0,Y 355.382,Z 287.082,A -85,B 0,C 180,E1 -14521.7,E2 -14521.7} C_VEL
LIN {X 0,Y 351.572,Z 266.466,A -85,B 0,C 180,E1 -14522.568,E2 -14522.568} C_VEL
LIN {X 0,Y 342.269,Z 246.321,A -85,B 0,C 180,E1 -14524.057,E2 -14524.057} C_VEL
LIN {X 0,Y 338.81,Z 238.969,A -85,B 0,C 180,E1 -14524.651,E2 -14524.651} C_VEL
LIN {X 0,Y 335.74,Z 227.698,A -85,B 0,C 180,E1 -14527.69,E2 -14527.69} C_VEL
LIN {X 0,Y 333.661,Z 220.547,A -85,B 0,C 180,E1 -14529.735,E2 -14529.735} C_VEL
LIN {X 0,Y 333.657,Z 220.547,A -85,B 0,C 180,E1 -14532.505,E2 -14532.505} C_VEL
LIN {X 0,Y 333.597,Z 220.556,A -85,B 0,C 180,E1 -14535.955,E2 -14535.955} C_VEL
LIN {X 0,Y 333.652,Z 220.542,A -85,B 0,C 180,E1 -14539.313,E2 -14539.313} C_VEL
LIN {X 0,Y 333.652,Z 220.543,A -85,B 0,C 180,E1 -14542.349,E2 -14542.349} C_VEL
LIN {X 0,Y 333.669,Z 220.54,A -85,B 0,C 180,E1 -14545.341,E2 -14545.341} C_VEL
LIN {X 0,Y 333.694,Z 220.538,A -85,B 0,C 180,E1 -14549.638,E2 -14549.638} C_VEL
LIN {X 0,Y 333.738,Z 220.533,A -85,B 0,C 180,E1 -14552.401,E2 -14552.401} C_VEL
LIN {X 0,Y 333.719,Z 220.54,A -85,B 0,C 180,E1 -14555.09,E2 -14555.09} C_VEL
LIN {X 0,Y 333.666,Z 220.523,A -85,B 0,C 180,E1 -14559.018,E2 -14559.018} C_VEL
LIN {X 0,Y 333.787,Z 220.533,A -85,B 0,C 180,E1 -14561.589,E2 -14561.589} C_VEL
LIN {X 0,Y 333.801,Z 220.533,A -85,B 0,C 180,E1 -14565.577,E2 -14565.577} C_VEL
LIN {X 0,Y 333.826,Z 220.525,A -85,B 0,C 180,E1 -14569.078,E2 -14569.078} C_VEL
LIN {X 0,Y 333.999,Z 220.502,A -85,B 0,C 180,E1 -14572.747,E2 -14572.747} C_VEL
LIN {X 0,Y 333.803,Z 220.525,A -85,B 0,C 180,E1 -14575.169,E2 -14575.169} C_VEL
LIN {X 0,Y 334.1,Z 220.496,A -85,B 0,C 180,E1 -14577.589,E2 -14577.589} C_VEL
LIN {X 0,Y 334.241,Z 220.467,A -85,B 0,C 180,E1 -14580,E2 -14580} C_VEL
LIN {X 0,Y 334.1,Z 220.492,A -85,B 0,C 180,E1 -14582.411,E2 -14582.411} C_VEL
LIN {X 0,Y 333.986,Z 220.504,A -85,B 0,C 180,E1 -14586.662,E2 -14586.662} C_VEL
LIN {X 0,Y 333.844,Z 220.524,A -85,B 0,C 180,E1 -14589.696,E2 -14589.696} C_VEL
LIN {X 0,Y 333.79,Z 220.527,A -85,B 0,C 180,E1 -14593.392,E2 -14593.392} C_VEL
LIN {X 0,Y 333.739,Z 220.532,A -85,B 0,C 180,E1 -14597.147,E2 -14597.147} C_VEL
LIN {X 0,Y 333.724,Z 220.536,A -85,B 0,C 180,E1 -14599.691,E2 -14599.691} C_VEL
LIN {X 0,Y 333.664,Z 220.543,A -85,B 0,C 180,E1 -14603.591,E2 -14603.591} C_VEL
LIN {X 0,Y 333.73,Z 220.51,A -85,B 0,C 180,E1 -14606.247,E2 -14606.247} C_VEL
LIN {X 0,Y 333.706,Z 220.542,A -85,B 0,C 180,E1 -14608.973,E2 -14608.973} C_VEL
LIN {X 0,Y 333.639,Z 220.551,A -85,B 0,C 180,E1 -14612.588,E2 -14612.588} C_VEL
LIN {X 0,Y 333.672,Z 220.544,A -85,B 0,C 180,E1 -14616.14,E2 -14616.14} C_VEL
LIN {X 0,Y 333.643,Z 220.544,A -85,B 0,C 180,E1 -14619.193,E2 -14619.193} C_VEL
LIN {X 0,Y 333.629,Z 220.546,A -85,B 0,C 180,E1 -14622.501,E2 -14622.501} C_VEL
LIN {X 0,Y 333.619,Z 220.551,A -85,B 0,C 180,E1 -14625.96,E2 -14625.96} C_VEL
LIN {X 0,Y 333.645,Z 220.552,A -85,B 0,C 180,E1 -14629.316,E2 -14629.316} C_VEL
LIN {X 0,Y 333.665,Z 220.547,A -85,B 0,C 180,E1 -14633.168,E2 -14633.168} C_VEL
LIN {X 0,Y 333.733,Z 220.67,A -85,B 0,C 180,E1 -14633.96,E2 -14633.96} C_VEL
LIN {X 0,Y 334.67,Z 224.06,A -85,B 0,C 180,E1 -14634.938,E2 -14634.938} C_VEL
LIN {X 0,Y 343.581,Z 240.814,A -85,B 0,C 180,E1 -14636.397,E2 -14636.397} C_VEL
LIN {X 0,Y 352.799,Z 259.953,A -85,B 0,C 180,E1 -14637.847,E2 -14637.847} C_VEL
LIN {X 0,Y 355.876,Z 267.209,A -85,B 0,C 180,E1 -14638.33,E2 -14638.33} C_VEL
LIN {X 0,Y 352.952,Z 370.4,A -85,B 0,C 180,E1 -14640.433,E2 -14640.433} C_VEL
LIN {X 0,Y 352.173,Z 390.839,A -85,B 0,C 180,E1 -14640.895,E2 -14640.895} C_VEL
LIN {X 0,Y 351.17,Z 405.696,A -85,B 0,C 180,E1 -14641.438,E2 -14641.438} C_VEL
LIN {X 0,Y 349.859,Z 420.503,A -85,B 0,C 180,E1 -14642.216,E2 -14642.216} C_VEL
LIN {X 0,Y 348.361,Z 434.24,A -85,B 0,C 180,E1 -14643.167,E2 -14643.167} C_VEL
LIN {X 0,Y 346.505,Z 447.485,A -85,B 0,C 180,E1 -14644.308,E2 -14644.308} C_VEL
LIN {X 0,Y 344.385,Z 460.942,A -85,B 0,C 180,E1 -14645.752,E2 -14645.752} C_VEL
LIN {X 0,Y 342.329,Z 472.785,A -85,B 0,C 180,E1 -14647.303,E2 -14647.303} C_VEL
LIN {X 0,Y 340.238,Z 484.267,A -85,B 0,C 180,E1 -14649.126,E2 -14649.126} C_VEL
LIN {X 0,Y 338.127,Z 495.062,A -85,B 0,C 180,E1 -14651.206,E2 -14651.206} C_VEL
LIN {X 0,Y 336.381,Z 504.019,A -85,B 0,C 180,E1 -14653.305,E2 -14653.305} C_VEL
LIN {X 0,Y 335.008,Z 511.438,A -85,B 0,C 180,E1 -14655.42,E2 -14655.42} C_VEL
LIN {X 0,Y 334.089,Z 516.771,A -85,B 0,C 180,E1 -14657.24,E2 -14657.24} C_VEL
LIN {X 0,Y 333.131,Z 522.586,A -85,B 0,C 180,E1 -14659.67,E2 -14659.67} C_VEL
LIN {X 0,Y 332.704,Z 526.026,A -85,B 0,C 180,E1 -14661.497,E2 -14661.497} C_VEL
LIN {X 0,Y 332.309,Z 529.511,A -85,B 0,C 180,E1 -14663.93,E2 -14663.93} C_VEL
LIN {X 0,Y 332.074,Z 531.814,A -85,B 0,C 180,E1 -14666.36,E2 -14666.36} C_VEL
LIN {X 0,Y 331.959,Z 532.991,A -85,B 0,C 180,E1 -14668.787,E2 -14668.787} C_VEL
LIN {X 0,Y 331.96,Z 533.005,A -85,B 0,C 180,E1 -14671.213,E2 -14671.213} C_VEL
LIN {X 0,Y 332.072,Z 531.888,A -85,B 0,C 180,E1 -14673.64,E2 -14673.64} C_VEL
LIN {X 0,Y 332.312,Z 529.391,A -85,B 0,C 180,E1 -14676.282,E2 -14676.282} C_VEL
LIN {X 0,Y 332.808,Z 525.155,A -85,B 0,C 180,E1 -14679.113,E2 -14679.113} C_VEL
LIN {X 0,Y 333.515,Z 520.101,A -85,B 0,C 180,E1 -14681.548,E2 -14681.548} C_VEL
LIN {X 0,Y 334.709,Z 513.621,A -85,B 0,C 180,E1 -14683.973,E2 -14683.973} C_VEL
LIN {X 0,Y 335.901,Z 506.631,A -85,B 0,C 180,E1 -14686.094,E2 -14686.094} C_VEL
LIN {X 0,Y 337.534,Z 498.213,A -85,B 0,C 180,E1 -14688.199,E2 -14688.199} C_VEL
LIN {X 0,Y 339.449,Z 488.074,A -85,B 0,C 180,E1 -14690.291,E2 -14690.291} C_VEL
LIN {X 0,Y 341.19,Z 478.93,A -85,B 0,C 180,E1 -14691.876,E2 -14691.876} C_VEL
LIN {X 0,Y 343.459,Z 466.402,A -85,B 0,C 180,E1 -14693.676,E2 -14693.676} C_VEL
LIN {X 0,Y 345.481,Z 454.123,A -85,B 0,C 180,E1 -14695.128,E2 -14695.128} C_VEL
LIN {X 0,Y 347.547,Z 440.692,A -85,B 0,C 180,E1 -14696.415,E2 -14696.415} C_VEL
LIN {X 0,Y 349.244,Z 426.773,A -85,B 0,C 180,E1 -14697.489,E2 -14697.489} C_VEL
LIN {X 0,Y 350.692,Z 412.122,A -85,B 0,C 180,E1 -14698.362,E2 -14698.362} C_VEL
LIN {X 0,Y 351.497,Z 401.978,A -85,B 0,C 180,E1 -14698.825,E2 -14698.825} C_VEL
LIN {X 0,Y 351.188,Z 398.182,A -85,B 0,C 180,E1 -14699.026,E2 -14699.026} C_VEL
LIN {X 0,Y 346.876,Z 386.414,A -85,B 0,C 180,E1 -14699.857,E2 -14699.857} C_VEL
LIN {X 0,Y 346.471,Z 382.561,A -85,B 0,C 180,E1 -14700.001,E2 -14700.001} C_VEL
LIN {X 0,Y 349.883,Z 272.175,A -85,B 0,C 180,E1 -14702.277,E2 -14702.277} C_VEL
LIN {X 0,Y 349.761,Z 268.892,A -85,B 0,C 180,E1 -14702.368,E2 -14702.368} C_VEL
LIN {X 0,Y 341.632,Z 251.136,A -85,B 0,C 180,E1 -14703.682,E2 -14703.682} C_VEL
LIN {X 0,Y 333.118,Z 234.626,A -85,B 0,C 180,E1 -14705.096,E2 -14705.096} C_VEL
LIN {X 0,Y 327.385,Z 224.07,A -85,B 0,C 180,E1 -14706.097,E2 -14706.097} C_VEL
LIN {X 0,Y 326.611,Z 221.423,A -85,B 0,C 180,E1 -14706.987,E2 -14706.987} C_VEL
LIN {X 0,Y 326.589,Z 221.422,A -85,B 0,C 180,E1 -14710.208,E2 -14710.208} C_VEL
LIN {X 0,Y 326.573,Z 221.432,A -85,B 0,C 180,E1 -14713.522,E2 -14713.522} C_VEL
LIN {X 0,Y 326.582,Z 221.416,A -85,B 0,C 180,E1 -14717.026,E2 -14717.026} C_VEL
LIN {X 0,Y 326.63,Z 221.419,A -85,B 0,C 180,E1 -14720.767,E2 -14720.767} C_VEL
LIN {X 0,Y 326.608,Z 221.422,A -85,B 0,C 180,E1 -14724.48,E2 -14724.48} C_VEL
LIN {X 0,Y 326.602,Z 221.408,A -85,B 0,C 180,E1 -14727.455,E2 -14727.455} C_VEL
LIN {X 0,Y 326.656,Z 221.412,A -85,B 0,C 180,E1 -14730.34,E2 -14730.34} C_VEL
LIN {X 0,Y 326.684,Z 221.412,A -85,B 0,C 180,E1 -14734.516,E2 -14734.516} C_VEL
LIN {X 0,Y 326.64,Z 221.418,A -85,B 0,C 180,E1 -14738.545,E2 -14738.545} C_VEL
LIN {X 0,Y 326.738,Z 221.402,A -85,B 0,C 180,E1 -14741.177,E2 -14741.177} C_VEL
LIN {X 0,Y 326.756,Z 221.397,A -85,B 0,C 180,E1 -14745.433,E2 -14745.433} C_VEL
LIN {X 0,Y 326.763,Z 221.404,A -85,B 0,C 180,E1 -14748.839,E2 -14748.839} C_VEL
LIN {X 0,Y 326.959,Z 221.384,A -85,B 0,C 180,E1 -14752.59,E2 -14752.59} C_VEL
LIN {X 0,Y 326.77,Z 221.398,A -85,B 0,C 180,E1 -14755.065,E2 -14755.065} C_VEL
LIN {X 0,Y 327.04,Z 221.371,A -85,B 0,C 180,E1 -14757.537,E2 -14757.537} C_VEL
LIN {X 0,Y 327.192,Z 221.344,A -85,B 0,C 180,E1 -14760,E2 -14760} C_VEL
LIN {X 0,Y 327.04,Z 221.372,A -85,B 0,C 180,E1 -14762.463,E2 -14762.463} C_VEL
LIN {X 0,Y 326.982,Z 221.38,A -85,B 0,C 180,E1 -14766.169,E2 -14766.169} C_VEL
LIN {X 0,Y 326.798,Z 221.4,A -85,B 0,C 180,E1 -14769.907,E2 -14769.907} C_VEL
LIN {X 0,Y 326.752,Z 221.403,A -85,B 0,C 180,E1 -14773.686,E2 -14773.686} C_VEL
LIN {X 0,Y 326.692,Z 221.407,A -85,B 0,C 180,E1 -14777.528,E2 -14777.528} C_VEL
LIN {X 0,Y 326.658,Z 221.423,A -85,B 0,C 180,E1 -14780.135,E2 -14780.135} C_VEL
LIN {X 0,Y 326.645,Z 221.424,A -85,B 0,C 180,E1 -14784.129,E2 -14784.129} C_VEL
LIN {X 0,Y 326.679,Z 221.419,A -85,B 0,C 180,E1 -14786.858,E2 -14786.858} C_VEL
LIN {X 0,Y 326.636,Z 221.424,A -85,B 0,C 180,E1 -14790.612,E2 -14790.612} C_VEL
LIN {X 0,Y 326.603,Z 221.424,A -85,B 0,C 180,E1 -14794.02,E2 -14794.02} C_VEL
LIN {X 0,Y 326.622,Z 221.423,A -85,B 0,C 180,E1 -14797.239,E2 -14797.239} C_VEL
LIN {X 0,Y 326.572,Z 221.408,A -85,B 0,C 180,E1 -14801.132,E2 -14801.132} C_VEL
LIN {X 0,Y 326.524,Z 221.435,A -85,B 0,C 180,E1 -14804.744,E2 -14804.744} C_VEL
LIN {X 0,Y 326.591,Z 221.425,A -85,B 0,C 180,E1 -14808.158,E2 -14808.158} C_VEL
LIN {X 0,Y 326.63,Z 221.53,A -85,B 0,C 180,E1 -14809.527,E2 -14809.527} C_VEL
LIN {X 0,Y 329.739,Z 232.195,A -85,B 0,C 180,E1 -14812.638,E2 -14812.638} C_VEL
LIN {X 0,Y 331.588,Z 238.898,A -85,B 0,C 180,E1 -14814.475,E2 -14814.475} C_VEL
LIN {X 0,Y 341.938,Z 260.395,A -85,B 0,C 180,E1 -14816.229,E2 -14816.229} C_VEL
LIN {X 0,Y 346.194,Z 270.25,A -85,B 0,C 180,E1 -14816.934,E2 -14816.934} C_VEL
LIN {X 0,Y 349.456,Z 289.089,A -85,B 0,C 180,E1 -14817.728,E2 -14817.728} C_VEL
LIN {X 0,Y 345.783,Z 405.176,A -85,B 0,C 180,E1 -14820.136,E2 -14820.136} C_VEL
LIN {X 0,Y 344.743,Z 420.616,A -85,B 0,C 180,E1 -14820.666,E2 -14820.666} C_VEL
LIN {X 0,Y 343.141,Z 435.531,A -85,B 0,C 180,E1 -14821.397,E2 -14821.397} C_VEL
LIN {X 0,Y 341.48,Z 449.276,A -85,B 0,C 180,E1 -14822.312,E2 -14822.312} C_VEL
LIN {X 0,Y 339.545,Z 462.401,A -85,B 0,C 180,E1 -14823.411,E2 -14823.411} C_VEL
LIN {X 0,Y 337.38,Z 475.127,A -85,B 0,C 180,E1 -14824.721,E2 -14824.721} C_VEL
LIN {X 0,Y 335.076,Z 488.006,A -85,B 0,C 180,E1 -14826.351,E2 -14826.351} C_VEL
LIN {X 0,Y 333.019,Z 498.548,A -85,B 0,C 180,E1 -14827.957,E2 -14827.957} C_VEL
LIN {X 0,Y 331.115,Z 508.78,A -85,B 0,C 180,E1 -14829.824,E2 -14829.824} C_VEL
LIN {X 0,Y 329.144,Z 518.551,A -85,B 0,C 180,E1 -14831.965,E2 -14831.965} C_VEL
LIN {X 0,Y 327.634,Z 526.712,A -85,B 0,C 180,E1 -14834.128,E2 -14834.128} C_VEL
LIN {X 0,Y 326.542,Z 533.464,A -85,B 0,C 180,E1 -14836.306,E2 -14836.306} C_VEL
LIN {X 0,Y 325.6,Z 539.702,A -85,B 0,C 180,E1 -14838.799,E2 -14838.799} C_VEL
LIN {X 0,Y 325.139,Z 544.533,A -85,B 0,C 180,E1 -14841.298,E2 -14841.298} C_VEL
LIN {X 0,Y 324.923,Z 548.615,A -85,B 0,C 180,E1 -14844.248,E2 -14844.248} C_VEL
LIN {X 0,Y 324.847,Z 550.405,A -85,B 0,C 180,E1 -14846.279,E2 -14846.279} C_VEL
LIN {X 0,Y 324.828,Z 551.577,A -85,B 0,C 180,E1 -14848.76,E2 -14848.76} C_VEL
LIN {X 0,Y 324.828,Z 551.574,A -85,B 0,C 180,E1 -14851.24,E2 -14851.24} C_VEL
LIN {X 0,Y 324.848,Z 550.391,A -85,B 0,C 180,E1 -14853.721,E2 -14853.721} C_VEL
LIN {X 0,Y 324.893,Z 548.05,A -85,B 0,C 180,E1 -14856.209,E2 -14856.209} C_VEL
LIN {X 0,Y 325.139,Z 544.505,A -85,B 0,C 180,E1 -14858.703,E2 -14858.703} C_VEL
LIN {X 0,Y 325.599,Z 539.667,A -85,B 0,C 180,E1 -14861.201,E2 -14861.201} C_VEL
LIN {X 0,Y 326.518,Z 533.41,A -85,B 0,C 180,E1 -14863.695,E2 -14863.695} C_VEL
LIN {X 0,Y 327.82,Z 525.557,A -85,B 0,C 180,E1 -14866.182,E2 -14866.182} C_VEL
LIN {X 0,Y 329.364,Z 517.212,A -85,B 0,C 180,E1 -14868.345,E2 -14868.345} C_VEL
LIN {X 0,Y 331.398,Z 507.167,A -85,B 0,C 180,E1 -14870.482,E2 -14870.482} C_VEL
LIN {X 0,Y 333.343,Z 496.896,A -85,B 0,C 180,E1 -14872.302,E2 -14872.302} C_VEL
LIN {X 0,Y 335.639,Z 484.661,A -85,B 0,C 180,E1 -14874.098,E2 -14874.098} C_VEL
LIN {X 0,Y 338.063,Z 471.042,A -85,B 0,C 180,E1 -14875.719,E2 -14875.719} C_VEL
LIN {X 0,Y 340.303,Z 457.392,A -85,B 0,C 180,E1 -14877.022,E2 -14877.022} C_VEL
LIN {X 0,Y 342.21,Z 443.502,A -85,B 0,C 180,E1 -14878.084,E2 -14878.084} C_VEL
LIN {X 0,Y 343.826,Z 428.689,A -85,B 0,C 180,E1 -14878.958,E2 -14878.958} C_VEL
LIN {X 0,Y 345.249,Z 412.702,A -85,B 0,C 180,E1 -14879.621,E2 -14879.621} C_VEL
LIN {X 0,Y 346.088,Z 396.66,A -85,B 0,C 180,E1 -14880.045,E2 -14880.045} C_VEL
LIN {X 0,Y 349.376,Z 289.616,A -85,B 0,C 180,E1 -14882.245,E2 -14882.245} C_VEL
LIN {X 0,Y 347.572,Z 278.102,A -85,B 0,C 180,E1 -14882.707,E2 -14882.707} C_VEL
LIN {X 0,Y 345.825,Z 269.272,A -85,B 0,C 180,E1 -14883.105,E2 -14883.105} C_VEL
LIN {X 0,Y 336.722,Z 249.39,A -85,B 0,C 180,E1 -14884.615,E2 -14884.615} C_VEL
LIN {X 0,Y 331.512,Z 238.616,A -85,B 0,C 180,E1 -14885.554,E2 -14885.554} C_VEL
LIN {X 0,Y 328.014,Z 226.12,A -85,B 0,C 180,E1 -14889.072,E2 -14889.072} C_VEL
LIN {X 0,Y 326.609,Z 221.428,A -85,B 0,C 180,E1 -14890.476,E2 -14890.476} C_VEL
LIN {X 0,Y 326.568,Z 221.429,A -85,B 0,C 180,E1 -14893.523,E2 -14893.523} C_VEL
LIN {X 0,Y 326.579,Z 221.424,A -85,B 0,C 180,E1 -14897.026,E2 -14897.026} C_VEL
LIN {X 0,Y 326.63,Z 221.419,A -85,B 0,C 180,E1 -14900.767,E2 -14900.767} C_VEL
LIN {X 0,Y 326.608,Z 221.417,A -85,B 0,C 180,E1 -14904.48,E2 -14904.48} C_VEL
LIN {X 0,Y 326.61,Z 221.417,A -85,B 0,C 180,E1 -14907.456,E2 -14907.456} C_VEL
LIN {X 0,Y 326.656,Z 221.413,A -85,B 0,C 180,E1 -14910.341,E2 -14910.341} C_VEL
LIN {X 0,Y 326.684,Z 221.416,A -85,B 0,C 180,E1 -14914.516,E2 -14914.516} C_VEL
LIN {X 0,Y 326.612,Z 221.398,A -85,B 0,C 180,E1 -14918.543,E2 -14918.543} C_VEL
LIN {X 0,Y 326.738,Z 221.407,A -85,B 0,C 180,E1 -14921.177,E2 -14921.177} C_VEL
LIN {X 0,Y 326.756,Z 221.409,A -85,B 0,C 180,E1 -14925.433,E2 -14925.433} C_VEL
LIN {X 0,Y 326.762,Z 221.404,A -85,B 0,C 180,E1 -14928.839,E2 -14928.839} C_VEL
LIN {X 0,Y 326.951,Z 221.379,A -85,B 0,C 180,E1 -14932.59,E2 -14932.59} C_VEL
LIN {X 0,Y 326.77,Z 221.402,A -85,B 0,C 180,E1 -14935.065,E2 -14935.065} C_VEL
LIN {X 0,Y 327.04,Z 221.374,A -85,B 0,C 180,E1 -14937.537,E2 -14937.537} C_VEL
LIN {X 0,Y 327.193,Z 221.344,A -85,B 0,C 180,E1 -14940,E2 -14940} C_VEL
LIN {X 0,Y 327.041,Z 221.371,A -85,B 0,C 180,E1 -14942.463,E2 -14942.463} C_VEL
LIN {X 0,Y 326.953,Z 221.379,A -85,B 0,C 180,E1 -14946.654,E2 -14946.654} C_VEL
LIN {X 0,Y 326.799,Z 221.401,A -85,B 0,C 180,E1 -14949.907,E2 -14949.907} C_VEL
LIN {X 0,Y 326.752,Z 221.406,A -85,B 0,C 180,E1 -14953.686,E2 -14953.686} C_VEL
LIN {X 0,Y 326.692,Z 221.412,A -85,B 0,C 180,E1 -14957.528,E2 -14957.528} C_VEL
LIN {X 0,Y 326.65,Z 221.416,A -85,B 0,C 180,E1 -14960.136,E2 -14960.136} C_VEL
LIN {X 0,Y 326.643,Z 221.415,A -85,B 0,C 180,E1 -14964.13,E2 -14964.13} C_VEL
LIN {X 0,Y 326.68,Z 221.391,A -85,B 0,C 180,E1 -14966.858,E2 -14966.858} C_VEL
LIN {X 0,Y 326.634,Z 221.42,A -85,B 0,C 180,E1 -14970.612,E2 -14970.612} C_VEL
LIN {X 0,Y 326.602,Z 221.42,A -85,B 0,C 180,E1 -14974.02,E2 -14974.02} C_VEL
LIN {X 0,Y 326.623,Z 221.42,A -85,B 0,C 180,E1 -14977.239,E2 -14977.239} C_VEL
LIN {X 0,Y 326.574,Z 221.426,A -85,B 0,C 180,E1 -14981.132,E2 -14981.132} C_VEL
LIN {X 0,Y 326.553,Z 221.43,A -85,B 0,C 180,E1 -14984.749,E2 -14984.749} C_VEL
LIN {X 0,Y 326.574,Z 221.43,A -85,B 0,C 180,E1 -14988.155,E2 -14988.155} C_VEL
LIN {X 0,Y 326.597,Z 221.419,A -85,B 0,C 180,E1 -14991.389,E2 -14991.389} C_VEL
LIN {X 0,Y 326.646,Z 221.456,A -85,B 0,C 180,E1 -14993.201,E2 -14993.201} C_VEL
LIN {X 0,Y 327.514,Z 224.409,A -85,B 0,C 180,E1 -14994.056,E2 -14994.056} C_VEL
LIN {X 0,Y 337.794,Z 243.45,A -85,B 0,C 180,E1 -14995.803,E2 -14995.803} C_VEL
LIN {X 0,Y 346.783,Z 262.175,A -85,B 0,C 180,E1 -14997.268,E2 -14997.268} C_VEL
LIN {X 0,Y 349.846,Z 269.307,A -85,B 0,C 180,E1 -14997.763,E2 -14997.763} C_VEL
LIN {X 0,Y 346.32,Z 384.314,A -85,B 0,C 180,E1 -15000.145,E2 -15000.145} C_VEL
LIN {X 0,Y 345.381,Z 400.336,A -85,B 0,C 180,E1 -15000.642,E2 -15000.642} C_VEL
LIN {X 0,Y 344.16,Z 415.234,A -85,B 0,C 180,E1 -15001.347,E2 -15001.347} C_VEL
LIN {X 0,Y 342.741,Z 428.61,A -85,B 0,C 180,E1 -15002.194,E2 -15002.194} C_VEL
LIN {X 0,Y 340.807,Z 442.982,A -85,B 0,C 180,E1 -15003.352,E2 -15003.352} C_VEL
LIN {X 0,Y 338.795,Z 456.039,A -85,B 0,C 180,E1 -15004.67,E2 -15004.67} C_VEL
LIN {X 0,Y 336.623,Z 468.061,A -85,B 0,C 180,E1 -15006.14,E2 -15006.14} C_VEL
LIN {X 0,Y 334.628,Z 479.158,A -85,B 0,C 180,E1 -15007.788,E2 -15007.788} C_VEL
LIN {X 0,Y 332.564,Z 489.34,A -85,B 0,C 180,E1 -15009.593,E2 -15009.593} C_VEL
LIN {X 0,Y 330.574,Z 499.298,A -85,B 0,C 180,E1 -15011.725,E2 -15011.725} C_VEL
LIN {X 0,Y 328.835,Z 507.556,A -85,B 0,C 180,E1 -15013.869,E2 -15013.869} C_VEL
LIN {X 0,Y 327.485,Z 515.303,A -85,B 0,C 180,E1 -15016.346,E2 -15016.346} C_VEL
LIN {X 0,Y 326.354,Z 521.471,A -85,B 0,C 180,E1 -15018.825,E2 -15018.825} C_VEL
LIN {X 0,Y 325.66,Z 526.229,A -85,B 0,C 180,E1 -15021.312,E2 -15021.312} C_VEL
LIN {X 0,Y 325.241,Z 529.712,A -85,B 0,C 180,E1 -15023.798,E2 -15023.798} C_VEL
LIN {X 0,Y 325.005,Z 532.015,A -85,B 0,C 180,E1 -15026.281,E2 -15026.281} C_VEL
LIN {X 0,Y 324.867,Z 533.191,A -85,B 0,C 180,E1 -15028.76,E2 -15028.76} C_VEL
LIN {X 0,Y 324.867,Z 533.206,A -85,B 0,C 180,E1 -15031.24,E2 -15031.24} C_VEL
LIN {X 0,Y 325.003,Z 532.088,A -85,B 0,C 180,E1 -15033.719,E2 -15033.719} C_VEL
LIN {X 0,Y 325.231,Z 529.769,A -85,B 0,C 180,E1 -15036.265,E2 -15036.265} C_VEL
LIN {X 0,Y 325.637,Z 526.409,A -85,B 0,C 180,E1 -15038.689,E2 -15038.689} C_VEL
LIN {X 0,Y 326.333,Z 521.709,A -85,B 0,C 180,E1 -15041.176,E2 -15041.176} C_VEL
LIN {X 0,Y 327.472,Z 515.613,A -85,B 0,C 180,E1 -15043.655,E2 -15043.655} C_VEL
LIN {X 0,Y 328.831,Z 507.94,A -85,B 0,C 180,E1 -15046.131,E2 -15046.131} C_VEL
LIN {X 0,Y 330.499,Z 499.75,A -85,B 0,C 180,E1 -15048.279,E2 -15048.279} C_VEL
LIN {X 0,Y 332.452,Z 489.883,A -85,B 0,C 180,E1 -15050.414,E2 -15050.414} C_VEL
LIN {X 0,Y 334.447,Z 479.762,A -85,B 0,C 180,E1 -15052.225,E2 -15052.225} C_VEL
LIN {X 0,Y 336.748,Z 467.706,A -85,B 0,C 180,E1 -15054.014,E2 -15054.014} C_VEL
LIN {X 0,Y 338.834,Z 455.614,A -85,B 0,C 180,E1 -15055.492,E2 -15055.492} C_VEL
LIN {X 0,Y 340.973,Z 442.468,A -85,B 0,C 180,E1 -15056.799,E2 -15056.799} C_VEL
LIN {X 0,Y 342.594,Z 429.94,A -85,B 0,C 180,E1 -15057.819,E2 -15057.819} C_VEL
LIN {X 0,Y 344.13,Z 416.006,A -85,B 0,C 180,E1 -15058.716,E2 -15058.716} C_VEL
LIN {X 0,Y 345.372,Z 400.929,A -85,B 0,C 180,E1 -15059.442,E2 -15059.442} C_VEL
LIN {X 0,Y 346.351,Z 385.307,A -85,B 0,C 180,E1 -15059.936,E2 -15059.936} C_VEL
LIN {X 0,Y 346.471,Z 382.561,A -85,B 0,C 180,E1 -15060.001,E2 -15060.001} C_VEL
LIN {X 0,Y 346.192,Z 376.774,A -85,B 0,C 180,E1 -15060.182,E2 -15060.182} C_VEL
LIN {X 0,Y 341.804,Z 358.152,A -85,B 0,C 180,E1 -15061.053,E2 -15061.053} C_VEL
LIN {X 0,Y 341.356,Z 352.353,A -85,B 0,C 180,E1 -15061.235,E2 -15061.235} C_VEL
LIN {X 0,Y 343.895,Z 271.348,A -85,B 0,C 180,E1 -15062.934,E2 -15062.934} C_VEL
LIN {X 0,Y 335.817,Z 253.655,A -85,B 0,C 180,E1 -15064.286,E2 -15064.286} C_VEL
LIN {X 0,Y 326.213,Z 235.211,A -85,B 0,C 180,E1 -15065.942,E2 -15065.942} C_VEL
LIN {X 0,Y 321.563,Z 227.097,A -85,B 0,C 180,E1 -15066.771,E2 -15066.771} C_VEL
LIN {X 0,Y 320.113,Z 224.215,A -85,B 0,C 180,E1 -15067.08,E2 -15067.08} C_VEL
LIN {X 0,Y 319.567,Z 222.306,A -85,B 0,C 180,E1 -15067.777,E2 -15067.777} C_VEL
LIN {X 0,Y 319.523,Z 222.312,A -85,B 0,C 180,E1 -15071.596,E2 -15071.596} C_VEL
LIN {X 0,Y 319.513,Z 222.312,A -85,B 0,C 180,E1 -15075.261,E2 -15075.261} C_VEL
LIN {X 0,Y 319.531,Z 222.299,A -85,B 0,C 180,E1 -15078.712,E2 -15078.712} C_VEL
LIN {X 0,Y 319.578,Z 222.28,A -85,B 0,C 180,E1 -15082.342,E2 -15082.342} C_VEL
LIN {X 0,Y 319.556,Z 222.305,A -85,B 0,C 180,E1 -15085.123,E2 -15085.123} C_VEL
LIN {X 0,Y 319.565,Z 222.277,A -85,B 0,C 180,E1 -15089.057,E2 -15089.057} C_VEL
LIN {X 0,Y 319.604,Z 222.299,A -85,B 0,C 180,E1 -15092.498,E2 -15092.498} C_VEL
LIN {X 0,Y 319.6,Z 222.301,A -85,B 0,C 180,E1 -15095.303,E2 -15095.303} C_VEL
LIN {X 0,Y 319.591,Z 222.294,A -85,B 0,C 180,E1 -15098.047,E2 -15098.047} C_VEL
LIN {X 0,Y 319.683,Z 222.282,A -85,B 0,C 180,E1 -15100.962,E2 -15100.962} C_VEL
LIN {X 0,Y 319.724,Z 222.274,A -85,B 0,C 180,E1 -15105.276,E2 -15105.276} C_VEL
LIN {X 0,Y 319.75,Z 222.271,A -85,B 0,C 180,E1 -15109.872,E2 -15109.872} C_VEL
LIN {X 0,Y 319.918,Z 222.26,A -85,B 0,C 180,E1 -15112.426,E2 -15112.426} C_VEL
LIN {X 0,Y 319.739,Z 222.273,A -85,B 0,C 180,E1 -15114.956,E2 -15114.956} C_VEL
LIN {X 0,Y 319.984,Z 222.25,A -85,B 0,C 180,E1 -15117.482,E2 -15117.482} C_VEL
LIN {X 0,Y 320.144,Z 222.222,A -85,B 0,C 180,E1 -15120,E2 -15120} C_VEL
LIN {X 0,Y 319.984,Z 222.25,A -85,B 0,C 180,E1 -15122.518,E2 -15122.518} C_VEL
LIN {X 0,Y 319.936,Z 222.259,A -85,B 0,C 180,E1 -15126.306,E2 -15126.306} C_VEL
LIN {X 0,Y 319.83,Z 222.263,A -85,B 0,C 180,E1 -15128.848,E2 -15128.848} C_VEL
LIN {X 0,Y 319.674,Z 222.283,A -85,B 0,C 180,E1 -15132.7,E2 -15132.7} C_VEL
LIN {X 0,Y 319.693,Z 222.289,A -85,B 0,C 180,E1 -15135.296,E2 -15135.296} C_VEL
LIN {X 0,Y 319.668,Z 222.293,A -85,B 0,C 180,E1 -15139.255,E2 -15139.255} C_VEL
LIN {X 0,Y 319.564,Z 222.305,A -85,B 0,C 180,E1 -15143.32,E2 -15143.32} C_VEL
LIN {X 0,Y 319.629,Z 222.29,A -85,B 0,C 180,E1 -15146.088,E2 -15146.088} C_VEL
LIN {X 0,Y 319.584,Z 222.302,A -85,B 0,C 180,E1 -15148.934,E2 -15148.934} C_VEL
LIN {X 0,Y 319.533,Z 222.306,A -85,B 0,C 180,E1 -15151.862,E2 -15151.862} C_VEL
LIN {X 0,Y 319.574,Z 222.299,A -85,B 0,C 180,E1 -15155.543,E2 -15155.543} C_VEL
LIN {X 0,Y 319.567,Z 222.304,A -85,B 0,C 180,E1 -15158.009,E2 -15158.009} C_VEL
LIN {X 0,Y 319.52,Z 222.29,A -85,B 0,C 180,E1 -15161.597,E2 -15161.597} C_VEL
LIN {X 0,Y 319.486,Z 222.315,A -85,B 0,C 180,E1 -15165.258,E2 -15165.258} C_VEL
LIN {X 0,Y 319.544,Z 222.335,A -85,B 0,C 180,E1 -15168.715,E2 -15168.715} C_VEL
LIN {X 0,Y 322.861,Z 233.609,A -85,B 0,C 180,E1 -15172.12,E2 -15172.12} C_VEL
LIN {X 0,Y 324.32,Z 238.755,A -85,B 0,C 180,E1 -15173.556,E2 -15173.556} C_VEL
LIN {X 0,Y 333.222,Z 256.717,A -85,B 0,C 180,E1 -15175.133,E2 -15175.133} C_VEL
LIN {X 0,Y 340.485,Z 272.811,A -85,B 0,C 180,E1 -15176.374,E2 -15176.374} C_VEL
LIN {X 0,Y 343.373,Z 289.365,A -85,B 0,C 180,E1 -15177.096,E2 -15177.096} C_VEL
LIN {X 0,Y 340.379,Z 384.862,A -85,B 0,C 180,E1 -15179.096,E2 -15179.096} C_VEL
LIN {X 0,Y 339.468,Z 407.375,A -85,B 0,C 180,E1 -15179.608,E2 -15179.608} C_VEL
LIN {X 0,Y 338.329,Z 422.787,A -85,B 0,C 180,E1 -15180.183,E2 -15180.183} C_VEL
LIN {X 0,Y 336.653,Z 437.681,A -85,B 0,C 180,E1 -15180.964,E2 -15180.964} C_VEL
LIN {X 0,Y 334.786,Z 451.944,A -85,B 0,C 180,E1 -15181.969,E2 -15181.969} C_VEL
LIN {X 0,Y 332.661,Z 465.298,A -85,B 0,C 180,E1 -15183.155,E2 -15183.155} C_VEL
LIN {X 0,Y 330.227,Z 478.73,A -85,B 0,C 180,E1 -15184.641,E2 -15184.641} C_VEL
LIN {X 0,Y 327.894,Z 490.97,A -85,B 0,C 180,E1 -15186.305,E2 -15186.305} C_VEL
LIN {X 0,Y 325.659,Z 502.032,A -85,B 0,C 180,E1 -15188.121,E2 -15188.121} C_VEL
LIN {X 0,Y 323.465,Z 513.006,A -85,B 0,C 180,E1 -15190.32,E2 -15190.32} C_VEL
LIN {X 0,Y 321.597,Z 522.05,A -85,B 0,C 180,E1 -15192.514,E2 -15192.514} C_VEL
LIN {X 0,Y 320.02,Z 530.622,A -85,B 0,C 180,E1 -15195.08,E2 -15195.08} C_VEL
LIN {X 0,Y 319.088,Z 536.569,A -85,B 0,C 180,E1 -15197.276,E2 -15197.276} C_VEL
LIN {X 0,Y 318.282,Z 542.083,A -85,B 0,C 180,E1 -15199.826,E2 -15199.826} C_VEL
LIN {X 0,Y 317.914,Z 546.258,A -85,B 0,C 180,E1 -15202.378,E2 -15202.378} C_VEL
LIN {X 0,Y 317.767,Z 549.186,A -85,B 0,C 180,E1 -15204.925,E2 -15204.925} C_VEL
LIN {X 0,Y 317.743,Z 550.933,A -85,B 0,C 180,E1 -15207.465,E2 -15207.465} C_VEL
LIN {X 0,Y 317.779,Z 551.531,A -85,B 0,C 180,E1 -15210,E2 -15210} C_VEL
LIN {X 0,Y 317.744,Z 550.924,A -85,B 0,C 180,E1 -15212.535,E2 -15212.535} C_VEL
LIN {X 0,Y 317.763,Z 549.165,A -85,B 0,C 180,E1 -15215.075,E2 -15215.075} C_VEL
LIN {X 0,Y 317.914,Z 546.23,A -85,B 0,C 180,E1 -15217.622,E2 -15217.622} C_VEL
LIN {X 0,Y 318.281,Z 542.051,A -85,B 0,C 180,E1 -15220.174,E2 -15220.174} C_VEL
LIN {X 0,Y 319.079,Z 536.523,A -85,B 0,C 180,E1 -15222.724,E2 -15222.724} C_VEL
LIN {X 0,Y 320.136,Z 529.49,A -85,B 0,C 180,E1 -15225.274,E2 -15225.274} C_VEL
LIN {X 0,Y 321.831,Z 520.752,A -85,B 0,C 180,E1 -15227.801,E2 -15227.801} C_VEL
LIN {X 0,Y 323.784,Z 511.477,A -85,B 0,C 180,E1 -15229.99,E2 -15229.99} C_VEL
LIN {X 0,Y 325.589,Z 502.105,A -85,B 0,C 180,E1 -15231.848,E2 -15231.848} C_VEL
LIN {X 0,Y 328.074,Z 489.824,A -85,B 0,C 180,E1 -15233.849,E2 -15233.849} C_VEL
LIN {X 0,Y 330.432,Z 477.363,A -85,B 0,C 180,E1 -15235.511,E2 -15235.511} C_VEL
LIN {X 0,Y 332.92,Z 463.582,A -85,B 0,C 180,E1 -15236.992,E2 -15236.992} C_VEL
LIN {X 0,Y 335.035,Z 449.818,A -85,B 0,C 180,E1 -15238.182,E2 -15238.182} C_VEL
LIN {X 0,Y 336.904,Z 435.007,A -85,B 0,C 180,E1 -15239.183,E2 -15239.183} C_VEL
LIN {X 0,Y 338.502,Z 419.959,A -85,B 0,C 180,E1 -15239.929,E2 -15239.929} C_VEL
LIN {X 0,Y 339.657,Z 404.2,A -85,B 0,C 180,E1 -15240.459,E2 -15240.459} C_VEL
LIN {X 0,Y 343.166,Z 296.207,A -85,B 0,C 180,E1 -15242.736,E2 -15242.736} C_VEL
LIN {X 0,Y 343.227,Z 288.774,A -85,B 0,C 180,E1 -15242.91,E2 -15242.91} C_VEL
LIN {X 0,Y 340.202,Z 272.164,A -85,B 0,C 180,E1 -15243.648,E2 -15243.648} C_VEL
LIN {X 0,Y 330.426,Z 250.79,A -85,B 0,C 180,E1 -15245.329,E2 -15245.329} C_VEL
LIN {X 0,Y 324.202,Z 238.447,A -85,B 0,C 180,E1 -15246.46,E2 -15246.46} C_VEL
LIN {X 0,Y 320.826,Z 226.558,A -85,B 0,C 180,E1 -15249.941,E2 -15249.941} C_VEL
LIN {X 0,Y 319.539,Z 222.305,A -85,B 0,C 180,E1 -15251.285,E2 -15251.285} C_VEL
LIN {X 0,Y 319.487,Z 222.309,A -85,B 0,C 180,E1 -15254.742,E2 -15254.742} C_VEL
LIN {X 0,Y 319.555,Z 222.302,A -85,B 0,C 180,E1 -15258.396,E2 -15258.396} C_VEL
LIN {X 0,Y 319.578,Z 222.294,A -85,B 0,C 180,E1 -15261.993,E2 -15261.993} C_VEL
LIN {X 0,Y 319.555,Z 222.297,A -85,B 0,C 180,E1 -15265.123,E2 -15265.123} C_VEL
LIN {X 0,Y 319.569,Z 222.299,A -85,B 0,C 180,E1 -15269.056,E2 -15269.056} C_VEL
LIN {X 0,Y 319.603,Z 222.294,A -85,B 0,C 180,E1 -15272.498,E2 -15272.498} C_VEL
LIN {X 0,Y 319.597,Z 222.301,A -85,B 0,C 180,E1 -15275.304,E2 -15275.304} C_VEL
LIN {X 0,Y 319.595,Z 222.278,A -85,B 0,C 180,E1 -15279.4,E2 -15279.4} C_VEL
LIN {X 0,Y 319.651,Z 222.292,A -85,B 0,C 180,E1 -15282.073,E2 -15282.073} C_VEL
LIN {X 0,Y 319.725,Z 222.282,A -85,B 0,C 180,E1 -15286.008,E2 -15286.008} C_VEL
LIN {X 0,Y 319.745,Z 222.281,A -85,B 0,C 180,E1 -15289.873,E2 -15289.873} C_VEL
LIN {X 0,Y 319.905,Z 222.257,A -85,B 0,C 180,E1 -15292.426,E2 -15292.426} C_VEL
LIN {X 0,Y 319.739,Z 222.279,A -85,B 0,C 180,E1 -15294.956,E2 -15294.956} C_VEL
LIN {X 0,Y 319.984,Z 222.252,A -85,B 0,C 180,E1 -15297.482,E2 -15297.482} C_VEL
LIN {X 0,Y 320.144,Z 222.222,A -85,B 0,C 180,E1 -15300,E2 -15300} C_VEL
LIN {X 0,Y 319.984,Z 222.25,A -85,B 0,C 180,E1 -15302.518,E2 -15302.518} C_VEL
LIN {X 0,Y 319.914,Z 222.256,A -85,B 0,C 180,E1 -15306.642,E2 -15306.642} C_VEL
LIN {X 0,Y 319.746,Z 222.28,A -85,B 0,C 180,E1 -15310.128,E2 -15310.128} C_VEL
LIN {X 0,Y 319.725,Z 222.283,A -85,B 0,C 180,E1 -15314.724,E2 -15314.724} C_VEL
LIN {X 0,Y 319.683,Z 222.291,A -85,B 0,C 180,E1 -15319.038,E2 -15319.038} C_VEL
LIN {X 0,Y 319.554,Z 222.302,A -85,B 0,C 180,E1 -15323.321,E2 -15323.321} C_VEL
LIN {X 0,Y 319.613,Z 222.267,A -85,B 0,C 180,E1 -15326.09,E2 -15326.09} C_VEL
LIN {X 0,Y 319.585,Z 222.301,A -85,B 0,C 180,E1 -15328.934,E2 -15328.934} C_VEL
LIN {X 0,Y 319.527,Z 222.307,A -85,B 0,C 180,E1 -15331.862,E2 -15331.862} C_VEL
LIN {X 0,Y 319.576,Z 222.3,A -85,B 0,C 180,E1 -15335.544,E2 -15335.544} C_VEL
LIN {X 0,Y 319.553,Z 222.302,A -85,B 0,C 180,E1 -15338.011,E2 -15338.011} C_VEL
LIN {X 0,Y 319.522,Z 222.302,A -85,B 0,C 180,E1 -15341.598,E2 -15341.598} C_VEL
LIN {X 0,Y 319.512,Z 222.307,A -85,B 0,C 180,E1 -15344.739,E2 -15344.739} C_VEL
LIN {X 0,Y 319.558,Z 222.304,A -85,B 0,C 180,E1 -15347.018,E2 -15347.018} C_VEL
LIN {X 0,Y 319.545,Z 222.299,A -85,B 0,C 180,E1 -15350.372,E2 -15350.372} C_VEL
LIN {X 0,Y 319.564,Z 222.324,A -85,B 0,C 180,E1 -15352.423,E2 -15352.423} C_VEL
LIN {X 0,Y 320.324,Z 224.631,A -85,B 0,C 180,E1 -15353.117,E2 -15353.117} C_VEL
LIN {X 0,Y 329.872,Z 242.031,A -85,B 0,C 180,E1 -15354.818,E2 -15354.818} C_VEL
LIN {X 0,Y 337.744,Z 257.819,A -85,B 0,C 180,E1 -15356.159,E2 -15356.159} C_VEL
LIN {X 0,Y 343.808,Z 271.244,A -85,B 0,C 180,E1 -15357.168,E2 -15357.168} C_VEL
LIN {X 0,Y 340.608,Z 372.638,A -85,B 0,C 180,E1 -15359.291,E2 -15359.291} C_VEL
LIN {X 0,Y 339.789,Z 392.411,A -85,B 0,C 180,E1 -15359.768,E2 -15359.768} C_VEL
LIN {X 0,Y 338.646,Z 407.862,A -85,B 0,C 180,E1 -15360.376,E2 -15360.376} C_VEL
LIN {X 0,Y 337.139,Z 423.198,A -85,B 0,C 180,E1 -15361.243,E2 -15361.243} C_VEL
LIN {X 0,Y 335.511,Z 436.413,A -85,B 0,C 180,E1 -15362.221,E2 -15362.221} C_VEL
LIN {X 0,Y 333.51,Z 449.325,A -85,B 0,C 180,E1 -15363.398,E2 -15363.398} C_VEL
LIN {X 0,Y 331.252,Z 462.521,A -85,B 0,C 180,E1 -15364.892,E2 -15364.892} C_VEL
LIN {X 0,Y 329.162,Z 473.519,A -85,B 0,C 180,E1 -15366.395,E2 -15366.395} C_VEL
LIN {X 0,Y 327.005,Z 484.674,A -85,B 0,C 180,E1 -15368.239,E2 -15368.239} C_VEL
LIN {X 0,Y 324.646,Z 495.471,A -85,B 0,C 180,E1 -15370.395,E2 -15370.395} C_VEL
LIN {X 0,Y 322.75,Z 504.427,A -85,B 0,C 180,E1 -15372.578,E2 -15372.578} C_VEL
LIN {X 0,Y 321.156,Z 511.847,A -85,B 0,C 180,E1 -15374.776,E2 -15374.776} C_VEL
LIN {X 0,Y 320.209,Z 517.177,A -85,B 0,C 180,E1 -15376.676,E2 -15376.676} C_VEL
LIN {X 0,Y 319.144,Z 522.991,A -85,B 0,C 180,E1 -15379.212,E2 -15379.212} C_VEL
LIN {X 0,Y 318.633,Z 526.431,A -85,B 0,C 180,E1 -15381.118,E2 -15381.118} C_VEL
LIN {X 0,Y 318.16,Z 530.001,A -85,B 0,C 180,E1 -15383.736,E2 -15383.736} C_VEL
LIN {X 0,Y 317.938,Z 532.216,A -85,B 0,C 180,E1 -15386.198,E2 -15386.198} C_VEL
LIN {X 0,Y 317.778,Z 533.392,A -85,B 0,C 180,E1 -15388.733,E2 -15388.733} C_VEL
LIN {X 0,Y 317.778,Z 533.406,A -85,B 0,C 180,E1 -15391.267,E2 -15391.267} C_VEL
LIN {X 0,Y 317.936,Z 532.288,A -85,B 0,C 180,E1 -15393.802,E2 -15393.802} C_VEL
LIN {X 0,Y 318.166,Z 530.042,A -85,B 0,C 180,E1 -15396.341,E2 -15396.341} C_VEL
LIN {X 0,Y 318.611,Z 526.61,A -85,B 0,C 180,E1 -15398.882,E2 -15398.882} C_VEL
LIN {X 0,Y 319.333,Z 521.91,A -85,B 0,C 180,E1 -15401.424,E2 -15401.424} C_VEL
LIN {X 0,Y 320.531,Z 515.814,A -85,B 0,C 180,E1 -15403.956,E2 -15403.956} C_VEL
LIN {X 0,Y 321.985,Z 508.139,A -85,B 0,C 180,E1 -15406.484,E2 -15406.484} C_VEL
LIN {X 0,Y 323.733,Z 499.95,A -85,B 0,C 180,E1 -15408.675,E2 -15408.675} C_VEL
LIN {X 0,Y 325.776,Z 490.082,A -85,B 0,C 180,E1 -15410.852,E2 -15410.852} C_VEL
LIN {X 0,Y 327.85,Z 479.961,A -85,B 0,C 180,E1 -15412.697,E2 -15412.697} C_VEL
LIN {X 0,Y 330.245,Z 467.904,A -85,B 0,C 180,E1 -15414.518,E2 -15414.518} C_VEL
LIN {X 0,Y 332.413,Z 455.812,A -85,B 0,C 180,E1 -15416.021,E2 -15416.021} C_VEL
LIN {X 0,Y 334.65,Z 442.663,A -85,B 0,C 180,E1 -15417.348,E2 -15417.348} C_VEL
LIN {X 0,Y 336.331,Z 430.134,A -85,B 0,C 180,E1 -15418.384,E2 -15418.384} C_VEL
LIN {X 0,Y 337.918,Z 416.37,A -85,B 0,C 180,E1 -15419.283,E2 -15419.283} C_VEL
LIN {X 0,Y 339.231,Z 401.117,A -85,B 0,C 180,E1 -15420.029,E2 -15420.029} C_VEL
LIN {X 0,Y 340.239,Z 385.486,A -85,B 0,C 180,E1 -15420.531,E2 -15420.531} C_VEL
LIN {X 0,Y 341.356,Z 352.353,A -85,B 0,C 180,E1 -15421.235,E2 -15421.235} C_VEL
LIN {X 0,Y 340.956,Z 346.563,A -85,B 0,C 180,E1 -15421.416,E2 -15421.416} C_VEL
LIN {X 0,Y 336.819,Z 327.927,A -85,B 0,C 180,E1 -15422.31,E2 -15422.31} C_VEL
LIN {X 0,Y 336.39,Z 322.14,A -85,B 0,C 180,E1 -15422.501,E2 -15422.501} C_VEL
LIN {X 0,Y 337.89,Z 273.411,A -85,B 0,C 180,E1 -15423.549,E2 -15423.549} C_VEL
LIN {X 0,Y 329.524,Z 255.145,A -85,B 0,C 180,E1 -15425.001,E2 -15425.001} C_VEL
LIN {X 0,Y 319.841,Z 236.668,A -85,B 0,C 180,E1 -15426.74,E2 -15426.74} C_VEL
LIN {X 0,Y 313.527,Z 225.995,A -85,B 0,C 180,E1 -15427.915,E2 -15427.915} C_VEL
LIN {X 0,Y 312.835,Z 224.519,A -85,B 0,C 180,E1 -15428.078,E2 -15428.078} C_VEL
LIN {X 0,Y 312.502,Z 223.185,A -85,B 0,C 180,E1 -15428.568,E2 -15428.568} C_VEL
LIN {X 0,Y 312.49,Z 223.184,A -85,B 0,C 180,E1 -15432.43,E2 -15432.43} C_VEL
LIN {X 0,Y 312.479,Z 223.184,A -85,B 0,C 180,E1 -15436.03,E2 -15436.03} C_VEL
LIN {X 0,Y 312.505,Z 223.184,A -85,B 0,C 180,E1 -15439.873,E2 -15439.873} C_VEL
LIN {X 0,Y 312.536,Z 223.156,A -85,B 0,C 180,E1 -15442.616,E2 -15442.616} C_VEL
LIN {X 0,Y 312.515,Z 223.179,A -85,B 0,C 180,E1 -15446.31,E2 -15446.31} C_VEL
LIN {X 0,Y 312.54,Z 223.169,A -85,B 0,C 180,E1 -15450.349,E2 -15450.349} C_VEL
LIN {X 0,Y 312.597,Z 223.165,A -85,B 0,C 180,E1 -15454.064,E2 -15454.064} C_VEL
LIN {X 0,Y 312.582,Z 223.166,A -85,B 0,C 180,E1 -15457.528,E2 -15457.528} C_VEL
LIN {X 0,Y 312.632,Z 223.158,A -85,B 0,C 180,E1 -15461.656,E2 -15461.656} C_VEL
LIN {X 0,Y 312.687,Z 223.149,A -85,B 0,C 180,E1 -15465.686,E2 -15465.686} C_VEL
LIN {X 0,Y 312.695,Z 223.151,A -85,B 0,C 180,E1 -15469.641,E2 -15469.641} C_VEL
LIN {X 0,Y 312.859,Z 223.138,A -85,B 0,C 180,E1 -15472.254,E2 -15472.254} C_VEL
LIN {X 0,Y 312.709,Z 223.148,A -85,B 0,C 180,E1 -15474.842,E2 -15474.842} C_VEL
LIN {X 0,Y 312.985,Z 223.115,A -85,B 0,C 180,E1 -15478.713,E2 -15478.713} C_VEL
LIN {X 0,Y 312.985,Z 223.123,A -85,B 0,C 180,E1 -15481.287,E2 -15481.287} C_VEL
LIN {X 0,Y 312.709,Z 223.155,A -85,B 0,C 180,E1 -15485.158,E2 -15485.158} C_VEL
LIN {X 0,Y 312.846,Z 223.136,A -85,B 0,C 180,E1 -15487.746,E2 -15487.746} C_VEL
LIN {X 0,Y 312.662,Z 223.163,A -85,B 0,C 180,E1 -15491.671,E2 -15491.671} C_VEL
LIN {X 0,Y 312.693,Z 223.163,A -85,B 0,C 180,E1 -15494.888,E2 -15494.888} C_VEL
LIN {X 0,Y 312.624,Z 223.171,A -85,B 0,C 180,E1 -15499.237,E2 -15499.237} C_VEL
LIN {X 0,Y 312.54,Z 223.18,A -85,B 0,C 180,E1 -15502.789,E2 -15502.789} C_VEL
LIN {X 0,Y 312.597,Z 223.165,A -85,B 0,C 180,E1 -15505.936,E2 -15505.936} C_VEL
LIN {X 0,Y 312.541,Z 223.18,A -85,B 0,C 180,E1 -15509.65,E2 -15509.65} C_VEL
LIN {X 0,Y 312.515,Z 223.177,A -85,B 0,C 180,E1 -15513.689,E2 -15513.689} C_VEL
LIN {X 0,Y 312.532,Z 223.178,A -85,B 0,C 180,E1 -15517.384,E2 -15517.384} C_VEL
LIN {X 0,Y 312.485,Z 223.159,A -85,B 0,C 180,E1 -15520.71,E2 -15520.71} C_VEL
LIN {X 0,Y 312.448,Z 223.187,A -85,B 0,C 180,E1 -15524.21,E2 -15524.21} C_VEL
LIN {X 0,Y 312.522,Z 223.296,A -85,B 0,C 180,E1 -15527.911,E2 -15527.911} C_VEL
LIN {X 0,Y 315.638,Z 233.756,A -85,B 0,C 180,E1 -15531.197,E2 -15531.197} C_VEL
LIN {X 0,Y 316.968,Z 238.433,A -85,B 0,C 180,E1 -15532.565,E2 -15532.565} C_VEL
LIN {X 0,Y 324.453,Z 253.076,A -85,B 0,C 180,E1 -15533.957,E2 -15533.957} C_VEL
LIN {X 0,Y 332.322,Z 269.776,A -85,B 0,C 180,E1 -15535.362,E2 -15535.362} C_VEL
LIN {X 0,Y 335.025,Z 276.426,A -85,B 0,C 180,E1 -15535.847,E2 -15535.847} C_VEL
LIN {X 0,Y 337.415,Z 291.415,A -85,B 0,C 180,E1 -15536.495,E2 -15536.495} C_VEL
LIN {X 0,Y 333.725,Z 400.295,A -85,B 0,C 180,E1 -15538.808,E2 -15538.808} C_VEL
LIN {X 0,Y 332.799,Z 415.656,A -85,B 0,C 180,E1 -15539.284,E2 -15539.284} C_VEL
LIN {X 0,Y 331.345,Z 429.934,A -85,B 0,C 180,E1 -15539.928,E2 -15539.928} C_VEL
LIN {X 0,Y 329.707,Z 443.513,A -85,B 0,C 180,E1 -15540.763,E2 -15540.763} C_VEL
LIN {X 0,Y 327.695,Z 457.223,A -85,B 0,C 180,E1 -15541.848,E2 -15541.848} C_VEL
LIN {X 0,Y 325.273,Z 470.815,A -85,B 0,C 180,E1 -15543.191,E2 -15543.191} C_VEL
LIN {X 0,Y 322.894,Z 483.243,A -85,B 0,C 180,E1 -15544.714,E2 -15544.714} C_VEL
LIN {X 0,Y 320.496,Z 494.69,A -85,B 0,C 180,E1 -15546.41,E2 -15546.41} C_VEL
LIN {X 0,Y 318.27,Z 505.224,A -85,B 0,C 180,E1 -15548.293,E2 -15548.293} C_VEL
LIN {X 0,Y 316.395,Z 514.166,A -85,B 0,C 180,E1 -15550.2,E2 -15550.2} C_VEL
LIN {X 0,Y 314.513,Z 522.974,A -85,B 0,C 180,E1 -15552.443,E2 -15552.443} C_VEL
LIN {X 0,Y 313.005,Z 530.874,A -85,B 0,C 180,E1 -15554.904,E2 -15554.904} C_VEL
LIN {X 0,Y 311.845,Z 537.863,A -85,B 0,C 180,E1 -15557.638,E2 -15557.638} C_VEL
LIN {X 0,Y 311.106,Z 543.051,A -85,B 0,C 180,E1 -15560.246,E2 -15560.246} C_VEL
LIN {X 0,Y 310.83,Z 546.056,A -85,B 0,C 180,E1 -15562.203,E2 -15562.203} C_VEL
LIN {X 0,Y 310.683,Z 548.986,A -85,B 0,C 180,E1 -15564.809,E2 -15564.809} C_VEL
LIN {X 0,Y 310.666,Z 550.733,A -85,B 0,C 180,E1 -15567.407,E2 -15567.407} C_VEL
LIN {X 0,Y 310.689,Z 551.331,A -85,B 0,C 180,E1 -15570,E2 -15570} C_VEL
LIN {X 0,Y 310.666,Z 550.724,A -85,B 0,C 180,E1 -15572.593,E2 -15572.593} C_VEL
LIN {X 0,Y 310.722,Z 548.592,A -85,B 0,C 180,E1 -15575.616,E2 -15575.616} C_VEL
LIN {X 0,Y 310.83,Z 546.027,A -85,B 0,C 180,E1 -15577.797,E2 -15577.797} C_VEL
LIN {X 0,Y 311.22,Z 541.847,A -85,B 0,C 180,E1 -15580.408,E2 -15580.408} C_VEL
LIN {X 0,Y 312.074,Z 536.319,A -85,B 0,C 180,E1 -15583.015,E2 -15583.015} C_VEL
LIN {X 0,Y 313.231,Z 529.286,A -85,B 0,C 180,E1 -15585.619,E2 -15585.619} C_VEL
LIN {X 0,Y 315.001,Z 520.547,A -85,B 0,C 180,E1 -15588.201,E2 -15588.201} C_VEL
LIN {X 0,Y 317.06,Z 511.272,A -85,B 0,C 180,E1 -15590.433,E2 -15590.433} C_VEL
LIN {X 0,Y 318.941,Z 502.01,A -85,B 0,C 180,E1 -15592.306,E2 -15592.306} C_VEL
LIN {X 0,Y 321.338,Z 490.646,A -85,B 0,C 180,E1 -15594.209,E2 -15594.209} C_VEL
LIN {X 0,Y 323.756,Z 478.384,A -85,B 0,C 180,E1 -15595.904,E2 -15595.904} C_VEL
LIN {X 0,Y 326.319,Z 464.906,A -85,B 0,C 180,E1 -15597.409,E2 -15597.409} C_VEL
LIN {X 0,Y 328.65,Z 450.472,A -85,B 0,C 180,E1 -15598.702,E2 -15598.702} C_VEL
LIN {X 0,Y 330.563,Z 436.051,A -85,B 0,C 180,E1 -15599.711,E2 -15599.711} C_VEL
LIN {X 0,Y 332.198,Z 421.427,A -85,B 0,C 180,E1 -15600.469,E2 -15600.469} C_VEL
LIN {X 0,Y 333.486,Z 405.406,A -85,B 0,C 180,E1 -15601.041,E2 -15601.041} C_VEL
LIN {X 0,Y 337.156,Z 298.168,A -85,B 0,C 180,E1 -15603.34,E2 -15603.34} C_VEL
LIN {X 0,Y 337.253,Z 289.957,A -85,B 0,C 180,E1 -15603.534,E2 -15603.534} C_VEL
LIN {X 0,Y 334.542,Z 274.946,A -85,B 0,C 180,E1 -15604.22,E2 -15604.22} C_VEL
LIN {X 0,Y 325.202,Z 254.529,A -85,B 0,C 180,E1 -15605.879,E2 -15605.879} C_VEL
LIN {X 0,Y 318.792,Z 242.033,A -85,B 0,C 180,E1 -15607.054,E2 -15607.054} C_VEL
LIN {X 0,Y 316.904,Z 238.279,A -85,B 0,C 180,E1 -15607.419,E2 -15607.419} C_VEL
LIN {X 0,Y 314.017,Z 228.243,A -85,B 0,C 180,E1 -15610.469,E2 -15610.469} C_VEL
LIN {X 0,Y 312.523,Z 223.183,A -85,B 0,C 180,E1 -15612.141,E2 -15612.141} C_VEL
LIN {X 0,Y 312.468,Z 223.188,A -85,B 0,C 180,E1 -15616.032,E2 -15616.032} C_VEL
LIN {X 0,Y 312.492,Z 223.177,A -85,B 0,C 180,E1 -15619.291,E2 -15619.291} C_VEL
LIN {X 0,Y 312.537,Z 223.174,A -85,B 0,C 180,E1 -15622.617,E2 -15622.617} C_VEL
LIN {X 0,Y 312.515,Z 223.175,A -85,B 0,C 180,E1 -15626.311,E2 -15626.311} C_VEL
LIN {X 0,Y 312.544,Z 223.171,A -85,B 0,C 180,E1 -15630.35,E2 -15630.35} C_VEL
LIN {X 0,Y 312.597,Z 223.169,A -85,B 0,C 180,E1 -15634.064,E2 -15634.064} C_VEL
LIN {X 0,Y 312.536,Z 223.153,A -85,B 0,C 180,E1 -15637.525,E2 -15637.525} C_VEL
LIN {X 0,Y 312.631,Z 223.169,A -85,B 0,C 180,E1 -15641.656,E2 -15641.656} C_VEL
LIN {X 0,Y 312.687,Z 223.162,A -85,B 0,C 180,E1 -15645.686,E2 -15645.686} C_VEL
LIN {X 0,Y 312.691,Z 223.161,A -85,B 0,C 180,E1 -15649.642,E2 -15649.642} C_VEL
LIN {X 0,Y 312.846,Z 223.136,A -85,B 0,C 180,E1 -15652.254,E2 -15652.254} C_VEL
LIN {X 0,Y 312.709,Z 223.155,A -85,B 0,C 180,E1 -15654.842,E2 -15654.842} C_VEL
LIN {X 0,Y 312.985,Z 223.122,A -85,B 0,C 180,E1 -15658.713,E2 -15658.713} C_VEL
LIN {X 0,Y 312.986,Z 223.119,A -85,B 0,C 180,E1 -15661.287,E2 -15661.287} C_VEL
LIN {X 0,Y 312.71,Z 223.15,A -85,B 0,C 180,E1 -15665.158,E2 -15665.158} C_VEL
LIN {X 0,Y 312.847,Z 223.134,A -85,B 0,C 180,E1 -15667.747,E2 -15667.747} C_VEL
LIN {X 0,Y 312.662,Z 223.16,A -85,B 0,C 180,E1 -15671.672,E2 -15671.672} C_VEL
LIN {X 0,Y 312.694,Z 223.16,A -85,B 0,C 180,E1 -15674.888,E2 -15674.888} C_VEL
LIN {X 0,Y 312.603,Z 223.171,A -85,B 0,C 180,E1 -15679.225,E2 -15679.225} C_VEL
LIN {X 0,Y 312.52,Z 223.183,A -85,B 0,C 180,E1 -15682.781,E2 -15682.781} C_VEL
LIN {X 0,Y 312.592,Z 223.141,A -85,B 0,C 180,E1 -15685.934,E2 -15685.934} C_VEL
LIN {X 0,Y 312.541,Z 223.178,A -85,B 0,C 180,E1 -15689.651,E2 -15689.651} C_VEL
LIN {X 0,Y 312.515,Z 223.175,A -85,B 0,C 180,E1 -15693.689,E2 -15693.689} C_VEL
LIN {X 0,Y 312.522,Z 223.176,A -85,B 0,C 180,E1 -15697.386,E2 -15697.386} C_VEL
LIN {X 0,Y 312.486,Z 223.184,A -85,B 0,C 180,E1 -15700.71,E2 -15700.71} C_VEL
LIN {X 0,Y 312.47,Z 223.182,A -85,B 0,C 180,E1 -15704.207,E2 -15704.207} C_VEL
LIN {X 0,Y 312.483,Z 223.186,A -85,B 0,C 180,E1 -15707.919,E2 -15707.919} C_VEL
LIN {X 0,Y 312.491,Z 223.291,A -85,B 0,C 180,E1 -15711.632,E2 -15711.632} C_VEL
LIN {X 0,Y 312.915,Z 224.835,A -85,B 0,C 180,E1 -15712.089,E2 -15712.089} C_VEL
LIN {X 0,Y 320.377,Z 237.669,A -85,B 0,C 180,E1 -15713.482,E2 -15713.482} C_VEL
LIN {X 0,Y 329.626,Z 255.39,A -85,B 0,C 180,E1 -15715.136,E2 -15715.136} C_VEL
LIN {X 0,Y 337.79,Z 273.178,A -85,B 0,C 180,E1 -15716.55,E2 -15716.55} C_VEL
LIN {X 0,Y 334.751,Z 367.502,A -85,B 0,C 180,E1 -15718.562,E2 -15718.562} C_VEL
LIN {X 0,Y 333.743,Z 391.488,A -85,B 0,C 180,E1 -15719.117,E2 -15719.117} C_VEL
LIN {X 0,Y 332.675,Z 406.173,A -85,B 0,C 180,E1 -15719.68,E2 -15719.68} C_VEL
LIN {X 0,Y 331.159,Z 421.158,A -85,B 0,C 180,E1 -15720.5,E2 -15720.5} C_VEL
LIN {X 0,Y 329.503,Z 434.86,A -85,B 0,C 180,E1 -15721.496,E2 -15721.496} C_VEL
LIN {X 0,Y 327.439,Z 448.103,A -85,B 0,C 180,E1 -15722.692,E2 -15722.692} C_VEL
LIN {X 0,Y 325.054,Z 461.558,A -85,B 0,C 180,E1 -15724.208,E2 -15724.208} C_VEL
LIN {X 0,Y 322.827,Z 472.831,A -85,B 0,C 180,E1 -15725.756,E2 -15725.756} C_VEL
LIN {X 0,Y 321.108,Z 481.341,A -85,B 0,C 180,E1 -15727.14,E2 -15727.14} C_VEL
LIN {X 0,Y 318.908,Z 491.275,A -85,B 0,C 180,E1 -15729.016,E2 -15729.016} C_VEL
LIN {X 0,Y 316.78,Z 500.971,A -85,B 0,C 180,E1 -15731.235,E2 -15731.235} C_VEL
LIN {X 0,Y 314.917,Z 509.091,A -85,B 0,C 180,E1 -15733.482,E2 -15733.482} C_VEL
LIN {X 0,Y 313.621,Z 515.71,A -85,B 0,C 180,E1 -15735.73,E2 -15735.73} C_VEL
LIN {X 0,Y 312.37,Z 521.877,A -85,B 0,C 180,E1 -15738.318,E2 -15738.318} C_VEL
LIN {X 0,Y 311.593,Z 526.633,A -85,B 0,C 180,E1 -15740.916,E2 -15740.916} C_VEL
LIN {X 0,Y 311.057,Z 530.422,A -85,B 0,C 180,E1 -15743.792,E2 -15743.792} C_VEL
LIN {X 0,Y 310.873,Z 532.417,A -85,B 0,C 180,E1 -15746.111,E2 -15746.111} C_VEL
LIN {X 0,Y 310.692,Z 533.593,A -85,B 0,C 180,E1 -15748.704,E2 -15748.704} C_VEL
LIN {X 0,Y 310.692,Z 533.607,A -85,B 0,C 180,E1 -15751.296,E2 -15751.296} C_VEL
LIN {X 0,Y 310.869,Z 532.488,A -85,B 0,C 180,E1 -15753.889,E2 -15753.889} C_VEL
LIN {X 0,Y 311.104,Z 530.242,A -85,B 0,C 180,E1 -15756.485,E2 -15756.485} C_VEL
LIN {X 0,Y 311.573,Z 526.81,A -85,B 0,C 180,E1 -15759.085,E2 -15759.085} C_VEL
LIN {X 0,Y 312.344,Z 522.111,A -85,B 0,C 180,E1 -15761.683,E2 -15761.683} C_VEL
LIN {X 0,Y 313.602,Z 516.015,A -85,B 0,C 180,E1 -15764.271,E2 -15764.271} C_VEL
LIN {X 0,Y 315.129,Z 508.34,A -85,B 0,C 180,E1 -15766.853,E2 -15766.853} C_VEL
LIN {X 0,Y 316.979,Z 500.15,A -85,B 0,C 180,E1 -15769.088,E2 -15769.088} C_VEL
LIN {X 0,Y 319.137,Z 490.281,A -85,B 0,C 180,E1 -15771.306,E2 -15771.306} C_VEL
LIN {X 0,Y 321.383,Z 479.54,A -85,B 0,C 180,E1 -15773.298,E2 -15773.298} C_VEL
LIN {X 0,Y 323.804,Z 468.101,A -85,B 0,C 180,E1 -15775.039,E2 -15775.039} C_VEL
LIN {X 0,Y 326.037,Z 456.008,A -85,B 0,C 180,E1 -15776.569,E2 -15776.569} C_VEL
LIN {X 0,Y 328.345,Z 442.859,A -85,B 0,C 180,E1 -15777.918,E2 -15777.918} C_VEL
LIN {X 0,Y 330.257,Z 429.127,A -85,B 0,C 180,E1 -15779.06,E2 -15779.06} C_VEL
LIN {X 0,Y 331.959,Z 414.364,A -85,B 0,C 180,E1 -15780.01,E2 -15780.01} C_VEL
LIN {X 0,Y 333.237,Z 399.478,A -85,B 0,C 180,E1 -15780.715,E2 -15780.715} C_VEL
LIN {X 0,Y 334.217,Z 384.163,A -85,B 0,C 180,E1 -15781.185,E2 -15781.185} C_VEL
LIN {X 0,Y 336.39,Z 322.14,A -85,B 0,C 180,E1 -15782.501,E2 -15782.501} C_VEL
LIN {X 0,Y 335.927,Z 316.35,A -85,B 0,C 180,E1 -15782.695,E2 -15782.695} C_VEL
LIN {X 0,Y 331.718,Z 297.764,A -85,B 0,C 180,E1 -15783.639,E2 -15783.639} C_VEL
LIN {X 0,Y 331.438,Z 291.969,A -85,B 0,C 180,E1 -15783.82,E2 -15783.82} C_VEL
LIN {X 0,Y 331.923,Z 275.508,A -85,B 0,C 180,E1 -15784.185,E2 -15784.185} C_VEL
LIN {X 0,Y 323.95,Z 258.183,A -85,B 0,C 180,E1 -15785.618,E2 -15785.618} C_VEL
LIN {X 0,Y 315.187,Z 241.234,A -85,B 0,C 180,E1 -15787.25,E2 -15787.25} C_VEL
LIN {X 0,Y 307.662,Z 228.37,A -85,B 0,C 180,E1 -15788.707,E2 -15788.707} C_VEL
LIN {X 0,Y 305.998,Z 225.966,A -85,B 0,C 180,E1 -15789.03,E2 -15789.03} C_VEL
LIN {X 0,Y 305.564,Z 224.644,A -85,B 0,C 180,E1 -15789.194,E2 -15789.194} C_VEL
LIN {X 0,Y 305.472,Z 224.051,A -85,B 0,C 180,E1 -15789.475,E2 -15789.475} C_VEL
LIN {X 0,Y 305.439,Z 224.064,A -85,B 0,C 180,E1 -15793.651,E2 -15793.651} C_VEL
LIN {X 0,Y 305.458,Z 224.044,A -85,B 0,C 180,E1 -15797.412,E2 -15797.412} C_VEL
LIN {X 0,Y 305.504,Z 224.038,A -85,B 0,C 180,E1 -15801.602,E2 -15801.602} C_VEL
LIN {X 0,Y 305.458,Z 224.059,A -85,B 0,C 180,E1 -15804.886,E2 -15804.886} C_VEL
LIN {X 0,Y 305.446,Z 224.033,A -85,B 0,C 180,E1 -15808.355,E2 -15808.355} C_VEL
LIN {X 0,Y 305.516,Z 224.05,A -85,B 0,C 180,E1 -15811.113,E2 -15811.113} C_VEL
LIN {X 0,Y 305.566,Z 224.04,A -85,B 0,C 180,E1 -15814.087,E2 -15814.087} C_VEL
LIN {X 0,Y 305.494,Z 224.051,A -85,B 0,C 180,E1 -15818.402,E2 -15818.402} C_VEL
LIN {X 0,Y 305.584,Z 224.036,A -85,B 0,C 180,E1 -15821.217,E2 -15821.217} C_VEL
LIN {X 0,Y 305.642,Z 224.027,A -85,B 0,C 180,E1 -15825.349,E2 -15825.349} C_VEL
LIN {X 0,Y 305.631,Z 224.032,A -85,B 0,C 180,E1 -15829.399,E2 -15829.399} C_VEL
LIN {X 0,Y 305.802,Z 224.017,A -85,B 0,C 180,E1 -15832.074,E2 -15832.074} C_VEL
LIN {X 0,Y 305.68,Z 224.023,A -85,B 0,C 180,E1 -15834.723,E2 -15834.723} C_VEL
LIN {X 0,Y 305.952,Z 223.991,A -85,B 0,C 180,E1 -15838.684,E2 -15838.684} C_VEL
LIN {X 0,Y 305.952,Z 223.999,A -85,B 0,C 180,E1 -15841.316,E2 -15841.316} C_VEL
LIN {X 0,Y 305.835,Z 224.016,A -85,B 0,C 180,E1 -15846.598,E2 -15846.598} C_VEL
LIN {X 0,Y 305.697,Z 224.025,A -85,B 0,C 180,E1 -15849.261,E2 -15849.261} C_VEL
LIN {X 0,Y 305.581,Z 224.038,A -85,B 0,C 180,E1 -15853.296,E2 -15853.296} C_VEL
LIN {X 0,Y 305.587,Z 224.047,A -85,B 0,C 180,E1 -15856.02,E2 -15856.02} C_VEL
LIN {X 0,Y 305.571,Z 224.049,A -85,B 0,C 180,E1 -15859.445,E2 -15859.445} C_VEL
LIN {X 0,Y 305.484,Z 224.06,A -85,B 0,C 180,E1 -15863.042,E2 -15863.042} C_VEL
LIN {X 0,Y 305.542,Z 224.045,A -85,B 0,C 180,E1 -15866.227,E2 -15866.227} C_VEL
LIN {X 0,Y 305.491,Z 224.058,A -85,B 0,C 180,E1 -15869.05,E2 -15869.05} C_VEL
